	bGearOutMode                 :BOOL;
    fMasterSyncPosition           :LREAL;  
    fSlaveSyncPosition              :LREAL;  

	bReady                            :BOOL;  
    bStartSync		 	               :BOOL;	
	bInSync		 	                   :BOOL;	
    bBusy                               :BOOL;	
	bError				               :BOOL;		

END_STRUCT
END_TYPE

// ---- DUTs/06_Interface/FB_Interface/ST_RecY.TcDUT
TYPE ST_RecY : //
STRUCT
	bEnable		                        :BOOL;	
 
	bReady                            :BOOL;  
	bRecOK	 	                   :BOOL;	
	bError				               :BOOL;			
END_STRUCT
END_TYPE

// ---- DUTs/06_Interface/FB_Interface/ST_TenBuffer.TcDUT
TYPE ST_TenBuffer :  //张力FB 接口信号
STRUCT
   	bExecute			                        :BOOL;	
  

	bError                                       :BOOL;

	bReady                                      :BOOL;
	bStartSync		                             :BOOL;
	bInSync		                                 :BOOL;//同步状态

END_STRUCT
END_TYPE

// ---- DUTs/06_Interface/FB_Interface/ST_Tension_1.TcDUT
TYPE ST_Tension_1 :  //张力FB 接口信号
STRUCT
	fWindDiameter           :REAL;//放卷实时直径
    fDanserDegree           :REAL;//摆杆实时位置
   
   	bTenExecute		        :BOOL;	//张力使能
	bStudyExecute           :BOOL;  //摆杆学习开始     
   	fStudyDiameter          :REAL;  //摆杆学习时放卷直径
	
	bReady                    :BOOL;  //张力功能准备好
	bTensionOK		       :BOOL;	//张力使能OK

	bError			           :BOOL;	//张力出错
                         
END_STRUCT
END_TYPE

// ---- DUTs/06_Interface/Method/ST_Method.TcDUT
TYPE ST_Method :  //    方法
STRUCT

             AllTempTurnON                            :ST_MethodOut;//温控开
             AllTempTurnOFF                           :ST_MethodOut;//温控关
          
             AllRectLock                                  :ST_MethodOut;//纠偏外部锁定
             AllRectAuto                                  :ST_MethodOut;//纠偏自动
             AllRectManual                              :ST_MethodOut;//纠偏手动
             AllRectCenter                               :ST_MethodOut;//j纠偏居中

            // AllTen                                          :ST_MethodOut;
          

             AllGear                                        :ST_MethodOut;
             AllHome                                      :ST_MethodOut;


           // P1Ten                                             :ST_MethodOut;
           // P2Ten                                             :ST_MethodOut;
            //P3Ten                                             :ST_MethodOut;

            P1Pole                                            :ST_MethodOut;   
            P2Pole                                            :ST_MethodOut;   
            P3Pole                                            :ST_MethodOut;   
            P1GM                                             :ST_MethodOut;    
            P2GM                                             :ST_MethodOut;   


            P1CamIn                                        :ST_MethodOut;
            P2CamIn_U                                     :ST_MethodOut;
            P2CamIn_D                                     :ST_MethodOut;
            P3CamIn_U                                     :ST_MethodOut;
            P3CamIn_D                                     :ST_MethodOut;


          P4ShortTestHome                              :ST_MethodOut;  //短路测试
          P4StackHome                                    :ST_MethodOut; //叠片台
          P4CutSyncHome                                 :ST_MethodOut ;  //裁切同步
          P4NGHome                                       :ST_MethodOut ;  //NG料盒



END_STRUCT
END_TYPE

// ---- DUTs/06_Interface/Method/ST_MethodOut.TcDUT
TYPE ST_MethodOut :  //    方法
STRUCT
             Execute            :BOOL;  
             Done1               :BOOL;  
             Done2               :BOOL;  
             Error               :BOOL;

END_STRUCT
END_TYPE

// ---- DUTs/07_Name/ST_MotorName.TcDUT
TYPE ST_MotorName ://毛刷马达名称
STRUCT
	DDR_Dust:INT;//主驱辊除尘毛刷
	CuterBeltDust:INT;//裁切输送皮带除尘
	NGReverseBeltDust	:INT;//踢废倒装皮带除尘
	DedustBeltDust	:INT;//极片上表面除尘皮带除尘
	DedustReverseBeltDust	:INT;//极片下表面除尘倒装皮带除尘

   PoleBrushDust_U        :INT;     //极片上表面毛刷除尘**)
   PoleBrushDust_D        :INT;     //极片下表面毛刷除尘**)
   FeduanbeltDust1		  :INT;  //分段皮带1毛刷
   FeduanbeltDust2		  :INT;  //分段皮带2毛刷
   FeduanbeltDust3		  :INT;  //分段皮带3毛刷
   
END_STRUCT
END_TYPE

// ---- DUTs/07_Name/ST_NGMark.TcDUT
TYPE ST_NGMark :   //模切段NG标志位
STRUCT
	NGMark:ARRAY[1..30]	OF	BOOL	;	//[1]极片长度不良计数标志位,[2]极片宽度不良计数标志位,[3]R角不良计数标志位,[4]极耳不良计数标志位,[5]CIL宽不良计数标志位,[6]极片角度、边缘角度不良计数标志位,[7]尺寸其他不良,[8]接带不良计数标志位,[9]极片破损不良计数标志位,[10]划痕不良计数标志位,[11]亮斑不良计数标志位,[12]黑点不良计数标志位,[13]脏污不良计数标志位,[14]脱碳不良计数标志位,


	//NGMark[1]	:	BOOL	;	//	极片长度不良计数标志位
	//NGMark[2]	:	BOOL	;	//	极片宽度不良计数标志位
	//NGMark[3]	:	BOOL	;	//	R角不良计数标志位
	//NGMark[4]	:	BOOL	;	//	极耳不良计数标志位
	//NGMark[5]	:	BOOL	;	//	CIL宽不良计数标志位
	//NGMark[6]	:	BOOL	;	//	极片角度、边缘角度不良计数标志位
	//NGMark[7]	:	BOOL	;	//	尺寸其他不良
	//NGMark[8]	:	BOOL	;	//	接带不良计数标志位
	//NGMark[9]	:	BOOL	;	//	极片破损不良计数标志位
	//NGMark[10]	:	BOOL	;	//	划痕不良计数标志位
	//NGMark[11]	:	BOOL	;	//	亮斑不良计数标志位
	//NGMark[12]	:	BOOL	;	//	黑点不良计数标志位
	//NGMark[13]	:	BOOL	;	//	脏污不良计数标志位
	//NGMark[14]	:	BOOL	;	//	脱碳不良计数标志位




END_STRUCT
END_TYPE

// ---- DUTs/07_Name/ST_TableNo.TcDUT
TYPE ST_TableNo ://    凸轮表号
STRUCT
         Cuter	:UINT ;(*裁切切刀凸轮编号*)
		 CuterStop	:UINT ;(*裁切切刀停止凸轮编号*)
		 Mould	:UINT;(*模具切刀凸轮编号*)
		 MouldStop	:UINT;(*模具切刀停止凸轮编号*)
         Dirver	:UINT;(*主驱动凸轮编号*)
		 VirDirver:UINT;(*虚驱动凸轮编号*)
         VirBelt	:UINT;(*虚拟皮带凸轮编号*)
         NgPush	:UINT;(*NG踢料凸轮编号*)
		 NgPushStop	:UINT;(*NG踢料停止凸轮编号*)
         BufferLine	:UINT;(*极片缓存凸轮编号*)
		 CCDPress:UINT;(*CCD压片凸轮编号*)
		 BufferLine_1	:UINT;(*极片缓存凸轮编号*)
END_STRUCT
END_TYPE

// ---- DUTs/07_Name/ST_CylinderName.TcDUT
TYPE ST_CylinderName :   //气缸名称
STRUCT
Inflation_L	:INT;(*左放卷气胀轴气缸*)	
Inflation_R	:INT;(*右放卷气胀轴气缸*)	
BoardPressL	:INT;(*左接带压板气缸*)	
BoardPressR	:INT;(*右接带压板气缸*)	
DriverPressAux	:INT;(*辅助驱动压辊气缸*)	
CoderRollPress	:INT;(*编码器辊压辊气缸*)	
DriverPressDDR	:INT;(*主驱动压辊气缸*)	
NGRevBeltUpDown	:INT;(*踢废倒装皮带升降气缸*)	
NGRevBeltTension	:INT;(*踢废倒装皮带张紧气缸*)	
PoleBrushDustPush_U	:INT;(*极片上表面毛刷除尘升降缸*)	
PoleWindDustPush_U	:INT;(*极片上表面风刀除尘升降缸*)	
PoleBrushDustPush_D	:INT;(*极片下表面毛刷除尘升降缸*)	
PoleWindDustPush_D	:INT;(*极片下表面风刀除尘升降缸*)	
DustRevBeltUpDown	:INT;(*极片下表面除尘倒装皮带升降气缸*)	
NGBoxLock1	:INT;(*NG料盒归正气缸1*)	
NGBoxLock2	:INT;(*NG料盒归正气缸2*)	
WasteBoxPush	:INT;(*连续废料收集箱推料气缸*)	
END_STRUCT
END_TYPE

// ---- DUTs/07_Name/ST_VirAxisName.TcDUT
TYPE ST_VirAxisName :   //正极虚轴名称
STRUCT
 VirMain:INT;//模切虚拟主轴
 VirDriver:INT;//模切虚拟驱动辊
 VirBelt:INT;//模切虚拟皮带轴
  
END_STRUCT
END_TYPE

// ---- DUTs/06_Interface/FB_Interface/ST_Tension.TcDUT
TYPE ST_Tension :  //张力FB 接口信号
STRUCT
	fWindDiameter           :REAL;//放卷实时直径
    fDanserDegree           :REAL;//摆杆实时位置
   
   	bTenExecute		        :BOOL;	//张力使能
	bStudyExecute           :BOOL;  //摆杆学习开始     
   	fStudyDiameter          :REAL;  //摆杆学习时放卷直径
	
	bReady                    :BOOL;  //张力功能准备好
	bTensionOK		       :BOOL;	//张力使能OK

	bError			           :BOOL;	//张力出错
                         
END_STRUCT
END_TYPE

// ---- DUTs/09_保持型汇总/LocalProduction.TcDUT
TYPE  LocalProduction :
STRUCT
	OutFlag1:BOOL;(*产量计数标志1*)
	OutFlag2:BOOL;(*产量计数标志2*)
	NGFlag:ARRAY[1..50] OF BOOL;(*NG1计数标志*)

	RunFlag:BOOL;(*运行标志*)
	WaitFlag:BOOL;(*待料标志*)
	AlarmFlag:BOOL;(*故障标志*)
	DelDataAMBtn:BOOL;(*白班数据清除按钮*)
	DelDataPMBtn:BOOL;(*夜班数据清除按钮*)
	NowOutTotal:REAL;(*当前班次加工总数*)
	NowRate:REAL;(*当前班次良率*)
	HMI_NGClearAMBtn:ARRAY[1..50] OF BOOL;//白班NG类型计数清零
	HMI_NGClearPMBtn:ARRAY[1..50] OF BOOL;//夜班NG类型计数清零
	
//产能清零
	HMI_DelDataAMBtn			:BOOL;//白班产能清零
	HMI_DelDataPMBtn			:BOOL;//夜班产能清零
(*产能统计*)
	HMI_TodayTotal				:REAL;(*当天24H生产总数*)
	HMI_TodayOK					:REAL; (*当天24H生产OK总数*)
	HMI_TodayNG 				:REAL; (*当天24H生产NG总数*)
	
	HMI_HistoryTotal			:ARRAY[1..7 ] 	OF REAL ;(*历史每天24H生产总数ARRAY[1..7 ]*)
	HMI_HistoryOK				:ARRAY[1..7 ] 	OF REAL ;(*历史每天24H生产OK总数ARRAY[1..7 ]*)
	HMI_HistoryNG 				:ARRAY[1..7 ] 	OF REAL ; (*历史每天24H生产NG总数ARRAY[1..7 ]*)
	DayCountTotal				:REAL;(*白班产量合计*)
	NightCountTotal				:REAL;(*夜班产量合计*)
	SaveNowDay					:INT;
	SaveNowMonth				:INT;
	nDayRunTimeCnt				:ARRAY[8..19 ] 	OF UDINT;		(*白班运行时间统计*)
	nDayAlarmTimeCnt			:ARRAY[8..19 ] 	OF UDINT;		(*白班报警时间统计*)
	nDayWaitTimeCnt				:ARRAY[8..19 ] 	OF UDINT;		(*白班待料时间统计*)
	nNightRunTimeCnt			:ARRAY[0..23 ] OF UDINT;		(*夜班运行时间统计*)
	nNightAlarmTimeCnt			:ARRAY[0..23 ] OF UDINT;		(*夜班报警时间统计*)
	nNightWaitTimeCnt			:ARRAY[0..23 ] OF UDINT;		(*夜班待料时间统计*)
	HourTimeDayCount			:ARRAY[8..19 ] 	OF REAL;		(*白班每小时产量*)
	HourTimeNightCount			:ARRAY[0..23] 	OF REAL;		(*夜班每小时产量*)
	NgPerHourDayCount			:ARRAY[1..50 ] 	OF REAL;		(*白班1-30种类的不良分类*)
	NgPerHourNightCount			:ARRAY[1..50 ] 	OF REAL;		(*夜班1-30种类的不良分类*)
	HMI_TotalCount				:REAL;(*总产量*)
	HMI_OkCount					:REAL;(*OK产量*)
	HMI_NgCount					:REAL;(*Ng产量*)
	HMI_Qualified 				:REAL;(*良率*)
	HMI_NG_Qualified 			:REAL;(*不良率*)
	HMI_OEE							:REAL;//设备稼动率
	HMI_DayOkCount				:REAL;(*白班OK产量*)
	HMI_DayNgCount				:REAL;(*白班Ng产量*)
	HMI_DayQualified 			:REAL;(*白班良率*)
	HMI_DayNG_Qualified 		:REAL;(*白班不良率*)
	HMI_NightOkCount			:REAL;(*夜班OK产量*)
	HMI_NightNgCount			:REAL;(*夜班Ng产量*)
	HMI_NightQualified 			:REAL;(*夜班良率*)
	HMI_NightNG_Qualified 		:REAL;(*夜班不良率*)
	DayRunTimeTotal				:REAL;(*白班总运行时间合计*)
	NightRunTimeTotal			:REAL;(*夜班总运行时间合计*)
	DayAlarmTimeTotal			:REAL;(*白班总报警时间合计*)
	NightAlarmTimeTotal			:REAL;(*夜班总报警时间合计*)
	DayWaitTimeTotal			:REAL;(*白班总待料时间合计*)
	NightWaitTimeTotal			:REAL;(*夜班总待料时间合计*)
	RunTimeTotal				:REAL;(*总运行时间合计*)
	WaitTimeTotal				:REAL;(*总待料时间合计*)
	AlarmTimeTotal				:REAL;(*总报警时间合计*)
	(*历史数据变量汇总1-7天*)
	(*白班*)
	DayReadDayHistory			:ARRAY[1..7 ] 	OF INT;(*历史日*)
	DayReadMonthHistory			:ARRAY[1..7 ] 	OF INT;(*历史月*)
	DayCountTotalHistory		:ARRAY[1..7 ] 	OF REAL ;(*历史白班每天生产总数*)
	HMI_DayOkCountHistory		:ARRAY[1..7 ] 	OF REAL ;(*历史白班每天生产OK总数*)
	HMI_DayNgCountHistory		:ARRAY[1..7 ] 	OF REAL ;(*历史白班每天生产NG总数*)
	HMI_DayQualifiedHistory		:ARRAY[1..7 ] 	OF REAL ;  (*历史白班每天良率*)
	DayRunTimeTotalHistory		:ARRAY[1..7 ] 	OF REAL ;(*历史每天白板总运行时间合计*)
	DayWaitTimeTotalHistory		:ARRAY[1..7 ] 	OF REAL ;(*历史每天白板总待料时间合计*)
	DayAlarmTimeTotalHistory	:ARRAY[1..7 ] 	OF REAL ;(*历史每天白板总报警时间合计*)
	NgPerHourDayCountHistory	:ARRAY[1..7,1..50 ] 	OF REAL ;(*历史每天白班各类NG数量*)
	HourTimeDayCountHistory		:ARRAY[1..7,8..19 ] 	OF REAL ;(*历史每天白班每小时产量*)
	(*夜班*)
	NightCountTotalHistory		:ARRAY[1..7 ] 	OF REAL ;
	HMI_NightOkCountHistory		:ARRAY[1..7 ] 	OF REAL ;
	HMI_NightNgCountHistory		:ARRAY[1..7 ] 	OF REAL ;
	HMI_NightQualifiedHistory	:ARRAY[1..7 ] 	OF REAL ;
	NightRunTimeTotalHistory	:ARRAY[1..7 ] 	OF REAL ;
	NightWaitTimeTotalHistory	:ARRAY[1..7 ] 	OF REAL ;
	NightAlarmTimeTotalHistory	:ARRAY[1..7 ] 	OF REAL ;
	NgPerHourNightCountHistory	:ARRAY[1..7,1..50 ] 	OF REAL ;
	HourTimeNightCountHistory	:ARRAY[1..7,0..23] 	OF REAL ;
	(*历史数据变量汇总1-7天*)


(**********************************生产统计数据********************************************)
	DayRunTime_min:ARRAY[8..19] 	OF REAL;	(*白班每小时运行时间*)
	NightRunTime_min:ARRAY[0..23] 	OF REAL;	(*夜班每小时运行时间*)
	AllDayRunTime_min: REAL;	(*白班总运行时间*)
	AllNightRunTime_min: REAL;	(*夜班总运行时间*)

	DayWaitTime_min:ARRAY[8..19] 	OF REAL;	(*白班待料每小时时间*)
	NightWaitTime_min:ARRAY[0..23] 	OF REAL;	(*夜班待料每小时时间*)
	AllDayWaitTime_min: REAL;(*白班总待料时间*)
	AllNightWaitTime_min: REAL;(*夜班总待料时间*)

	DayAlmTime_min:ARRAY[8..19] 	OF REAL;	(*白班每小时报警时间*)
	NightAlmTime_min:ARRAY[0..23] OF REAL;	(*夜班每小时报警时间*)
	AllDayAlmTime_min: REAL;	(*白班总报警时间*)
	AllNightAlmTime_min: REAL;	(*夜班总报警时间*)

	DayBlockTime_min:ARRAY[0..23] 	OF REAL;(*白班每小时堵料时间*)
	NightBlockTime_min:ARRAY[0..23] 	OF REAL;(*夜班每小时堵料时间*)
	AllDayBlockTime_min: REAL;(*白班总堵料时间*)
	AllNightBlockTime_min: REAL;(*夜班总堵料时间*)
	
	HMINgClassCount_Day:ARRAY[1..50,0..23] 	OF REAL;(*白班每种NG类型每小时统计 ,,,NG类型，小时*)
	HMINgClassCount_Night:ARRAY[1..50,0..23] 	OF REAL;(*夜班每种NG类型每小时统计 ,,,NG类型，小时*)
	
	
	

	HisDayRunTime_min	:ARRAY[1..7,8..19 ] OF REAL ; (*历史白班每小时运行时间*)
	HisNightRunTime_min	:ARRAY[1..7,0..23 ] OF REAL ; (*历史夜班每小时运行时间*)
	HisAllDayRunTime_min:ARRAY[1..7] OF REAL ;	(*历史白班总运行时间*)
	HisAllNightRunTime_min:ARRAY[1..7 ] OF REAL ;	(*历史夜班总运行时间*)

	HisDayWaitTime_min	:ARRAY[1..7,8..19 ] OF REAL ; (*历史白班每小时待料时间*)
	HisNightWaitTime_min:ARRAY[1..7,0..23 ] OF REAL ; (*历史夜班每小时待料时间*)
	HisAllDayWaitTime_min:ARRAY[1..7] OF REAL ;	(*历史白班总待料时间*)
	HisAllNightWaitTime_min:ARRAY[1..7 ] OF REAL ;	(*历史夜班总待料时间*)

	HisDayAlmTime_min	:ARRAY[1..7,8..19 ] OF REAL ; (*历史白班每小时报警时间*)
	HisNightAlmTime_min	:ARRAY[1..7,0..23 ] OF REAL ; (*历史夜班每小时报警时间*)
	HisAllDayAlmTime_min:ARRAY[1..7] OF REAL ;	(*历史白班总报警时间*)
	HisAllNightAlmTime_min:ARRAY[1..7 ] OF REAL ;(*历史夜班总报警时间*)

	HisHMINgClassCount_Day:ARRAY[1..50,0..23,1..7] 	OF REAL;(*历史白班每种NG类型每小时统计,,,NG类型，小时，天*)
	HisHMINgClassCount_Night:ARRAY[1..50,0..23,1..7] 	OF REAL;(*历史夜班每种NG类型每小时统计,,,NG类型，小时，天*)

	
	HMI_TodayNGQualified:ARRAY[1..50] OF REAL;//当天白班各种NG类型NG率
	HMI_NightNGQualified:ARRAY[1..50] OF REAL;//当天夜班各种NG类型NG率	
	
	HMI_HisTodayNGQualified:ARRAY[1..50,1..7] OF REAL;//历史白班各种NG类型NG率
	HMI_HisNightNGQualified:ARRAY[1..50,1..7] OF REAL;//历史夜班各种NG类型NG率
	
END_STRUCT
END_TYPE

// ---- DUTs/09_保持型汇总/ST_Data.TcDUT
TYPE ST_Data :
STRUCT
	 AnBeltData:ARRAY[1..40]   OF  ST_BeltData;//正极皮带数据
	 CaBeltData:ARRAY[1..40]   OF  ST_BeltData;//负极皮带数据
	AnTabData:ARRAY[1..20]   OF  ST_TabData;//正极极耳数据
	CaTabData:ARRAY[1..20]   OF  ST_TabData;//负极极耳数据
	AnIntervalData:ARRAY[1..20]   OF  ST_IntervalData;//正极极耳间距数据
	CaIntervalData:ARRAY[1..20]   OF  ST_IntervalData;//负极极耳间距数据
	AnOffsetData:ARRAY[1..50]   OF  REAL;//正极主驱补偿数据
	CaOffsetData:ARRAY[1..50]   OF  REAL;//负极主驱补偿数据
	
	AnYellowPos:ARRAY [1..100] OF REAL;//正极黄标位置
	CaYellowPos:ARRAY [1..100] OF REAL;//负极黄标位置
	AnYellowMark:ARRAY [1..100] OF BOOL;//正极黄标标志--给到极片
	CaYellowMark:ARRAY [1..100] OF BOOL;//负极黄标标志--给到极片
	
	AnTapePos:ARRAY [1..100] OF REAL;//正极接带位置
	CaTapePos:ARRAY [1..100] OF REAL;//负极接带位置
	AnTapeMark:ARRAY [1..100] OF BOOL;//正极接带标志--给到极片
	CaTapeMark:ARRAY [1..100] OF BOOL;//负极接带标志--给到极片
	
	
	AnYellowJump_R:ARRAY [1..100] OF BOOL;//极片黄标R角跳切标志
	AnYellowJump_C:ARRAY [1..100] OF BOOL;//极片黄标裁切跳切标志
	AnTapeJump_R:ARRAY [1..100] OF BOOL;//极片接带R角跳切标志
	AnTapeJump_C:ARRAY [1..100] OF BOOL;//极片接带裁切跳切标志
	
	CaYellowJump_R:ARRAY [1..100] OF BOOL;//极片黄标R角跳切标志
	CaYellowJump_C:ARRAY [1..100] OF BOOL;//极片黄标裁切跳切标志
	CaTapeJump_R:ARRAY [1..100] OF BOOL;//极片接带R角跳切标志
	CaTapeJump_C:ARRAY [1..100] OF BOOL;//极片接带裁切跳切标志
			
END_STRUCT
END_TYPE

// ---- DUTs/09_保持型汇总/ST_Name.TcDUT
TYPE ST_Name :
STRUCT
(**轴**)
	AnAxisNo:      ST_AxisName;  //正极
	CaAxisNo:      ST_AxisName;//负极
	
    AnVirAxisNo:      ST_VirAxisName;//正极
	CaVirAxisNo:      ST_VirAxisName;//负极
	VirTimeWind:INT;//模切虚拟摆杆放卷轴 
(**气缸**)
	AnCYNo:        ST_CylinderName;//正极
	CaCYNo:        ST_CylinderName;//负极

(**电磁阀**)
	AnEVNo:        ST_ElectValveName;//正极
	CaEVNo:        ST_ElectValveName;//负极

(***纠偏**)
    AnRecNo:         ST_RecName;//正极
	CaRecNo:         ST_RecName;//负极

(***凸轮表号**)
	 AnTableNo:  ST_TableNo;// 正极
	 CaTableNo:  ST_TableNo;// 负极
	 
(***除尘电机号**)
	 AnMotorNo:  ST_MotorName;// 正极
	 CaMotorNo:  ST_MotorName;// 负极

(***数据工位号**)	 
	 AnBeltNo:ST_BeltNo;//正极
	 CaBeltNo:ST_BeltNo;//负极
	 AnTabNo:ST_TabNo;//正极
	 CaTabNo:ST_TabNo;//负极
	 AnIntervalNo:ST_IntervalNo;//正极
	 CaIntervalNo:ST_IntervalNo;//负极
END_STRUCT
END_TYPE

// ---- DUTs/09_保持型汇总/ST_Parameter.TcDUT
TYPE ST_Parameter :
STRUCT
	FanEn:BOOL;//风速仪屏蔽
	MaFanEn:BOOL;//风机平板
	AnPar: ST_ParProduct;   //正极工艺参数
	CaPar: ST_ParProduct;   //负极工艺参数
	parPublic:ST_PARpublic;//公共工艺参数
	
	parFilterAD            :ARRAY[1..MaxAINo] OF ST_ParFilterAD;
	parFilterDA            :ARRAY[1..2] OF ST_ParFilterDA;
	
	parDA                   :ARRAY[1..8] OF INT;   //模拟量输出
	iModeEN :                     IModeEN;//功能屏蔽

	  ////////////////////////////////////////////////////////////////////////////////////////////////////////////////断电保持中转变量////////////////////////////////////////////////////////////////////// 
	   	   
	 PoleData:ST_Data;	   
	   
	aAnDay_date: Day_date; //正极产能；
	aCaDay_date: Day_date; //负极产能；
	cCn_An:REAL;
	cCn_Ca:REAL;
		 
 	 YL_GVL2: ARRAY [1..60] OF DINT ;//内部预留；//  1、正极R角已经切的次数;  2、正极R角设置清废报警次数；3、负极R角已经切的次数;  4、负极R角设置清废报警次数；
	
(*产能统计*)	
	HMI_AnTodayNGClass_AM		:ARRAY[1..30 ] 	OF REAL;(*当天白班各类NG数量ARRAY[1..30 ]-----正极*)
	HMI_AnTodayNGClass_PM		:ARRAY[1..30 ] 	OF REAL;(*当天夜班各类NG数量ARRAY[1..30 ]-----正极*)
	HMI_AnTodayNG_AM:REAL;(*当天白班生产NG总数-----正极*)
	HMI_AnTodayNG_PM:REAL;(*当天夜班生产NG总数-----正极*)
	
	HMI_CaTodayNGClass_AM		:ARRAY[1..30 ] 	OF REAL;(*当天白班各类NG数量ARRAY[1..30 ]-----负极*)
	HMI_CaTodayNGClass_PM		:ARRAY[1..30 ] 	OF REAL;(*当天夜班各类NG数量ARRAY[1..30 ]-----负极*)
	HMI_CaTodayNG_AM:REAL;(*当天白班生产NG总数-----负极*)
	HMI_CaTodayNG_PM:REAL;(*当天夜班生产NG总数-----负极*)
	
	  iTargetTorque	                    	:ARRAY[1..2]OF INT;			                     (*单位为0.1%*) //最大为100

	CleanTimeHMIHour1:INT;//白班第一次清洁时间Hour\
	CleanTimeHMIMin1:INT;//白班第一次清洁时间Min
	CleanTimeHMIHour2:INT;//白班第二次清洁时间Hour
	CleanTimeHMIMin2:INT;//白班第二次清洁时间Min
	CleanTimeHMIHour3:INT;//夜班第一次清洁时间Hour
	CleanTimeHMIMin3:INT;//夜班第一次清洁时间Min
	CleanTimeHMIHour4:INT;//夜班第二次清洁时间Hour
	CleanTimeHMIMin4:INT;//夜班第二次清洁时间Ming
	CibangTimeHMIHour1:INT;//正极磁棒校验到期时间Hour
	CibangTimeHMIDay1:INT;//正极磁棒校验到期时间日
	CibangTimeHMIHour2:INT;//负极磁棒校验到期时间Hour
	CibangTimeHMIDay2:INT;//负极磁棒校验到期时间日	
	BrushTimeHMIHour1:INT;//正极毛刷清洁时间Hour
	BrushTimeHMIDay1:INT;//正极毛刷清洁时间Day
	BrushTimeHMIHour2:INT;//负极毛刷清洁时间Hour
	BrushTimeHMIDay2:INT;//负极毛刷清洁时间Day

(*****************************************************极耳基准20240101SJ*********************************************************************)	  

	bCompSel:BOOL;//补偿方案选择		
	
(***************************************************线扫20240219***********************************************************************)
	iLineScanSel:BOOL;//线扫结果控制模式
	
	  
(***************************************************4l连续黄标尾料检测***********************************************************************)
	fYellowMackLength1           :REAL;// 相邻黄标后边距离	
	  
END_STRUCT
END_TYPE

// ---- DUTs/30_Parameter/ST_DT_To_MQ_MES.TcDUT
TYPE ST_DT_To_MQ_MES  :
STRUCT
//PC写给PLC的-----先下发给叠台，叠台再和模切做通讯-------需要上料时PLC往该地址写入Error
PostiveCode1				:STRING(49);//正极左1条码		1
PostiveCode2				:STRING(49);//正极右2条码		2
NegativeCode1				:STRING(49);//负极左1条码		3
NegativeCode2				:STRING(49);//负极右2条码		4
Station1_Code				:STRING(49);//叠台1隔膜条码		5
Station2_Code				:STRING(49);//叠台2隔膜条码		6
Station3_Code				:STRING(49);//叠台3隔膜条码		7
Station1_BlueCode			:STRING(49);//叠台1l蓝胶条码		8
Station2_BlueCode			:STRING(49);//叠台2蓝胶条码		9
Station3_BlueCode			:STRING(49);//叠台3蓝胶条码		10
CellCode					:STRING(49);//后段二维码胶条码	11
BlueCode					:STRING(49);//后段蓝胶条码		12

//MES条码校验信号交互----PC_To_PLC
Mes_PcToPlc1:        BOOL;   //正极左1条码条码校验完成信号
Mes_PcToPlc2:        BOOL;   //正极右2条码校验完成信号
Mes_PcToPlc3:        BOOL;   //负极左1条码	校验完成信号
Mes_PcToPlc4:        BOOL;   //负极右2条码校验完成信号
Mes_PcToPlc5:        BOOL;   //叠台1隔膜条码校验完成信号
Mes_PcToPlc6:        BOOL;   //叠台2隔膜条码校验完成信号
Mes_PcToPlc7:        BOOL;   //叠台3隔膜条码校验完成信号
Mes_PcToPlc8:        BOOL;   //叠台1l蓝胶条码校验完成信号
Mes_PcToPlc9:        BOOL;   //叠台2蓝胶条码校验完成信号
Mes_PcToPlc10:        BOOL;  //叠台3蓝胶条码校验完成信号
Mes_PcToPlc11:        BOOL;   //后段二维码胶条码校验完成信号
Mes_PcToPlc12:        BOOL;   //后段蓝胶条码校验完成信号	

//MES条码校验信号交互----PLC_To_PC
MesClear_Pc1:        BOOL;   //正极左1换料信号清理
MesClear_Pc2:        BOOL;   //正极右2换料信号清理
MesClear_Pc3:        BOOL;   //负极左1换料信号清理
MesClear_Pc4:        BOOL;   //负极右2换料信号清理

END_STRUCT
END_TYPE

// ---- DUTs/30_Parameter/ST_MouldRecY.TcDUT
TYPE ST_MouldRecY :
STRUCT
		fRecBaseValue1                         :REAL:=5;//模具Y纠偏传感器基准值1(靠近大板)
		fRecBaseValue2							:REAL:=5;//模具Y纠偏传感器基准值2(远离大板)	
		fRectifyCoe                                 :REAL:=1;//纠偏系数	
		bRectifyDir                                 :BOOL;//纠偏方向
		fRecBaseRange                           :REAL:=0.2;//纠偏无效范围     注：纠偏量超出此值，才会进行动作。
		iMode                                        :INT:=1;//纠偏模式   1=单边纠偏；2=双边纠偏
		fRecAxisPos_H                             :REAL:=4;//纠偏电机上限
		fRecAxisPos_L                             :REAL:=4;//纠偏电机下限
END_STRUCT
END_TYPE

// ---- DUTs/30_Parameter/ST_MQ_To_DT_MES.TcDUT
TYPE ST_MQ_To_DT_MES  :
STRUCT
//PC写给PLC的-----先下发给叠台，叠台再和模切做通讯-------需要上料时PLC往该地址写入Error
PostiveCode1				:STRING(49);//正极左1条码		1
PostiveCode2				:STRING(49);//正极右2条码		2
NegativeCode1				:STRING(49);//负极左1条码		3
NegativeCode2				:STRING(49);//负极右2条码		4
Station1_Code				:STRING(49);//叠台1隔膜条码		5
Station2_Code				:STRING(49);//叠台2隔膜条码		6
Station3_Code				:STRING(49);//叠台3隔膜条码		7
Station1_BlueCode			:STRING(49);//叠台1l蓝胶条码		8
Station2_BlueCode			:STRING(49);//叠台2蓝胶条码		9
Station3_BlueCode			:STRING(49);//叠台3蓝胶条码		10
CellCode					:STRING(49);//后段二维码胶条码	11
BlueCode					:STRING(49);//后段蓝胶条码		12

//MES条码校验信号交互----PC_To_PLC
Mes_PcToPlc1:        BOOL;   //正极左1条码条码校验完成信号
Mes_PcToPlc2:        BOOL;   //正极右2条码校验完成信号
Mes_PcToPlc3:        BOOL;   //负极左1条码	校验完成信号
Mes_PcToPlc4:        BOOL;   //负极右2条码校验完成信号
Mes_PcToPlc5:        BOOL;   //叠台1隔膜条码校验完成信号
Mes_PcToPlc6:        BOOL;   //叠台2隔膜条码校验完成信号
Mes_PcToPlc7:        BOOL;   //叠台3隔膜条码校验完成信号
Mes_PcToPlc8:        BOOL;   //叠台1l蓝胶条码校验完成信号
Mes_PcToPlc9:        BOOL;   //叠台2蓝胶条码校验完成信号
Mes_PcToPlc10:        BOOL;  //叠台3蓝胶条码校验完成信号
Mes_PcToPlc11:        BOOL;   //后段二维码胶条码校验完成信号
Mes_PcToPlc12:        BOOL;   //后段蓝胶条码校验完成信号	

//MES条码校验信号交互----PLC_To_PC
Mes_PlcToPc1:        BOOL;   //正极左1换料信号
Mes_PlcToPc2:        BOOL;   //正极右2换料信号
Mes_PlcToPc3:        BOOL;   //负极左1换料信号
Mes_PlcToPc4:        BOOL;   //负极右2换料信号

END_STRUCT
END_TYPE

// ---- DUTs/30_Parameter/ST_ParFilterAD.TcDUT
TYPE ST_ParFilterAD :  //P1部分参数
STRUCT
	iLimitH             :REAL;//转换前高限值
	iLimitL             :REAL;//转换前低限值
	fRangeH         :REAL;//量程高限
	fRangeL          :REAL;//量程低限
	Out_Value        :REAL;//转换后

END_STRUCT
END_TYPE

// ---- DUTs/30_Parameter/ST_ParFilterDA.TcDUT
TYPE ST_ParFilterDA :  //P1部分参数
STRUCT
	X0:REAL;  //料带张力低限值g
	Y0:REAL;  //低限对应DA输出值
	X1:REAL; //料带张力高限值g
	Y1:REAL;//低限对应DA输出值
	bMode: BOOL;  //标定模式   TRUE为标定模式    
	iDAValue:REAL;//比例阀给定值     标定用
END_STRUCT
END_TYPE

// ---- DUTs/30_Parameter/ST_ParMachine.TcDUT
TYPE ST_ParMachine ://机械参数
STRUCT
       fMQDriverDiameter            :REAL:=71.62   ;//模切主驱辊直径
       fCuterDegDiameter				:REAL:=281.5   ;//裁切角度纠偏旋转半径
       fAuxDriverInDiameter         :REAL:=80   ;  //辅驱辊直径
	   fBelt1Scaling                      :REAL:=1   ;  //裁切皮带定长比例系数
	   fBelt2Scaling                      :REAL:=1   ;  //踢废倒装皮带定长比例系数
	   fBelt3Scaling                      :REAL:=1   ;  //上表面除尘皮带定长比例系数
	   fBelt4Scaling                      :REAL:=1   ;  //下表面除尘倒装皮带定长比例系数
	   fBelt5Scaling                      :REAL:=1   ;  //送料分段皮带1定长比例系数	   
	   fBelt6Scaling                      :REAL:=1   ;  //送料分段皮带2定长比例系数	   
	   fBelt7Scaling                      :REAL:=1   ;  //送料分段皮带3定长比例系数	  	   
//叠片主驱动  70
//叠片辅驱动  30
//NG皮带 46































END_STRUCT
END_TYPE

// ---- DUTs/30_Parameter/ST_MoQiePar.TcDUT
TYPE ST_MoQiePar :  //模切部分参数
STRUCT
(***张力参数*)
	TenCcw_WindL                            :BOOL;  //左放卷放卷方向
	TenCcw_WindR                            :BOOL;  //右放卷放卷方向
	bWindSelect								:BOOL;//放卷选择ON=使用左放卷
	WindPidSwitch                         :BOOL;  //放卷PID使能开关
	WindTenMinPos                      :REAL;//放卷摆杆最小角度
	WindTenMaxPos                     :REAL; //放卷摆杆最大角度
	WindTenBlancePos                  :REAL ;//放卷摆杆平衡角度
	WindTenTable                        :ARRAY[0..105,1..2]OF REAL;	//放卷摆杆采样数据
	
	TenCcw_AuxDriver                            :BOOL;  //辅驱放卷方向
	AuxDriverPidSwitch                         :BOOL;  //辅驱PID使能开关
	AuxDriverTenMinPos                      :REAL;//辅驱摆杆最小角度
	AuxDriverTenMaxPos                     :REAL; //辅驱摆杆最大角度
	AuxDriverTenBlancePos                  :REAL ;//辅驱摆杆平衡角度
	AuxDriverTenTable                        :ARRAY[0..105,1..2]OF REAL;	//辅驱摆杆采样数据		
	
	BufferPidSwitch                         :BOOL;  //缓存PID使能开关
	BufferMinPos                            :REAL;//缓存最小角度
	BufferMaxPos                           :REAL; //缓存最大角度
	BufferBlancePos                        :REAL ;//缓存平衡角度


   
END_STRUCT
END_TYPE

// ---- DUTs/30_Parameter/ST_ParProduct.TcDUT
TYPE ST_ParProduct ://工艺参数
STRUCT
(***HMI***)
	fYellowWidth :REAL:=25 ;    //黄标宽度
	fTapeWidth :REAL:=30 ;    //接带胶纸宽度
	fPoleWidth                          		  :REAL:=100 ;    //片宽
	fBeltSpacePos            :REAL:=280;//皮带运行定长
	
	//fCentreWidth_L								:REAL;//极耳中心_极片左侧宽度基准（程序内称左肩宽）
	//fCentreWidth_R								:REAL;//极耳中心_极片右侧宽度基准（程序内称右肩宽）
	fBlue_Mould                                :REAL;//蓝胶检测到模具倒角前的距离
	//iMould_Cuter                               :INT;//模具与裁切间的极耳个数
	fLineNG_Mould							   :REAL;//缺陷NG点到模具倒角前的距离
	bEarCheckMode                            :BOOL;   //极耳检测模式     FALSE:定长     TRUE：检测极耳
	fEarCheckLength                            :REAL;   //检测到极耳后走定长长度
	
	
	fFr_TenValuehmi									:REAL;//后摆杆张力比例阀大小HMI设置   单位%   范围：0-100
	fPressDDRhmi									:REAL;//主驱压辊比例阀大小HMI设置   单位%   范围：0-100
	
	iMouldCount1									:DINT;//前模具切刀计数
	iMouldCount2									:DINT;//后模具切刀计数
	iCuterCount									:DINT;//裁切切刀计数
	iMouldclear1                                 :BOOL;//前倒角模具切刀清零
	iMouldclear2                                 :BOOL;//后倒角模具切刀清零
	iCuterclear                                 :BOOL;//裁切切刀清零
	iMouldCountAlarm1						    :DINT;//前模具切刀计数报警
	iMouldCountAlarm2						    :DINT;//后模具切刀计数报警
	iCuterCountAlarm						     :DINT;//裁切切刀计数报警
	iCuterCountWarning							:DINT;//裁切切刀计数预警
	iCuterBarCode								:STRING(49);//切刀条码
	iReplaceCuterTime							:STRING(49);//换刀时间
	
	iMainVel                                  :UINT:=10;  //设置速度 PPM (最小值1,最大值200)          
	fMainHmiVel                                  :REAL;  //显示料带速度 M/min  
	fDiameterWarn_L:REAL;//左放卷卷径临界设置(警告)
	fDiameterWarn_R:REAL;//右放卷卷径临界设置(警告)
	fDiameterAlarm_L:REAL;//左放卷卷径临界设置(报警)
	fDiameterAlarm_R:REAL;//右放卷卷径临界设置(报警)
	
	MQ:ST_MoQiePar; (******放卷部分参数******)
	Rec:ST_MouldRecY;(******Y纠偏部分参数******)
	Machine: ST_ParMachine;   //机械参数常量   不允许外部改变
/////////////////////////////////////////////////////////////////////////////////////////////////CCD  R角闭环纠偏参数/////////////////////////////////////////////////////////////////////		
	Databace_R3:REAL;//CCD_R3 非极耳侧纵深基准正极5.6  负极2.6
	Databace_R4:REAL;//CCD_R4非极耳侧纵深基准正极5.6  负极2.6
	IntervalNum:UINT:=7; //片间距
	KI_Riao:REAL:=0.3;//比例系数		
	Limt_Max:REAL:=0.5; //最大补偿值
	Limt_Min:REAL:=-0.5;//最小补偿值
	TabSitebace:REAL;//基准肩宽
	TabWidthBace: REAL;//标准间距		
	AddAlarm:INT;
////////////////////////////////////////////////////////////////////////////////////////////////////////////////////////////////////////////////////////////////////////////////////////////////////		
(***内部使用**)
	fPoleWithOffset						:REAL; //主驱片宽补偿值（计算后）
	fMouldX_Offset						:REAL; //模具肩宽补偿值（计算后）
	fDegreeRectify						:REAL; //裁切角度纠偏值（计算后）
	fMouldY_Rectify						:REAL; //倒角深度纠偏值（计算后）
	
	
	fTension   							:REAL;//模切张力
	fSpeed								:REAL;//模切速度

//皮带齿轮比计算
	BeltDust1Great:REAL;//皮带1齿轮比计算系数
	BeltDust2Great:REAL;//皮带2齿轮比计算系数
	BeltDust3Great:REAL;//皮带3齿轮比计算系数

      

//新黄标、接带检测
	fLugBreadth:REAL:=59;//极耳宽度
	fCutBreadth:REAL:=22;//极耳边到切刀切点宽度---23.5+-1
	fYellowBreadth:REAL:=35;//黄标宽度
	fTapeBreadth:REAL:=35;//接带宽度
	
//初始卷径标定 ----demarcate
	rRoll_L:REAL:=1000;//缓存极片总长度(mm)
	rRollStartView:REAL;//放卷开始角度
        rRollFinishView:REAL;//放卷结束角度 
	rRollView :REAL;//放卷运动总角度  
	rRollDia:REAL;//初始卷径(计数输出)
	bDemarcateBtn:BOOL;//标定开始按钮

fTape_Mould                                :REAL;//接带检测到模具倒角前的距离	
fTape1_2                                :REAL;//前接带检到后接带检测的距离
(*****************************************************极耳基准20240101SJ*********************************************************************)	  

	fTabWidth: REAL;//极耳标准宽
	fDriverStanderBasePos: REAL;//极耳下降沿基准主驱凸轮位置
	fReadDriverPos3: REAL;//读取极耳下降沿主驱凸轮表位置
	bDriverStanderBasePosEN: BOOL;  //极耳大范围调整屏蔽	
	


END_STRUCT
END_TYPE

// ---- DUTs/30_Parameter/ST_ParPublic.TcDUT
TYPE ST_ParPublic :
STRUCT
		   fMainPos                   :REAL:=250;     //主轴关键点角度
		   //fBeltSpacePos            :REAL:=280;//皮带运行定长
END_STRUCT
END_TYPE

// ---- DUTs/30_Parameter/ST_ParTemperature.TcDUT
TYPE ST_ParTemperature ://   温控相关参数
STRUCT
   fTempSet                                   :REAL;// 设定温度温度(转换后)
   fTempOffset                               :REAL;// 设定温度温度(转换后);// 温度偏移

   fTempMax                                :REAL;     //温度高限设置

  fTempArea                               :REAL;     

END_STRUCT
END_TYPE

// ---- DUTs/31_其他辅助/ST_Timedata_2.TcDUT
TYPE ST_Timedata_2 :
STRUCT
	
	RunTime:ARRAY[0..25] OF UINT;//运行时间
    WaitTime:ARRAY[0..25] OF UINT;//待机时间
    AlmTime:ARRAY[0..25] OF UINT;//报警时间 	
    changeTime:ARRAY[0..25] OF UINT;//极片更换等待时间  	

	
END_STRUCT
END_TYPE

// ---- DUTs/32_系统/ST_SystemPart.TcDUT
TYPE ST_SystemPart ://系统功能块UDT
STRUCT
(***btn***)
	 btnStart                      :BOOL;  //面板启动
     btnStop                      :BOOL;  //面板停止
	 btnReset                     :BOOL;  //面板复位
     btnAuto                      :BOOL;//面板true=自动；false=手动
	 btnEstop                    :BOOL;//面板急停	 
	 
	 boStartLight                     :BOOL;           (***面板启动按钮灯***)
	 boResetLight                     :BOOL;           (***面板复位按钮灯***)
	 boStopLight                     :BOOL;           (***面板停止按钮灯***)
(***HMI*) 
	 hmiTenAll                    :BOOL;  //一键张力耦合
	 hmiDisTenAll                    :BOOL;  //一键张力解耦
	 hmiCamAll                    :BOOL;  //一键凸轮耦合
	 hmiDisCamAll                    :BOOL;  //一键凸轮解耦
	 hmiGoHome					:BOOL;//一键初始化(回原)
	 hmiClearBelt                 :BOOL;//一键清皮带(清除皮带上的料)
	 
	 hmiMQDriverOnce          :BOOL;  //模切驱动一片
	 hmiMQCutOnce             :BOOL;  //模切裁切一片 
	 
	 
(**Status**)
	 Homed						:BOOL;//初始化完成
	 Homeing					:BOOL;//初始化进行中
     Autoing                     :BOOL;   //自动运行中
	 Manuling                   :BOOL;  //手动运行中
	 Stoping                     :BOOL;   //停止中
	 Alarming                   :BOOL;   //报警中
	 bErrorStop                :BOOL;//报警停机

     bAutoCondition1         :BOOL;//自动准备好(初步)
	 bAutoCondition2         :BOOL;//自动准备好(张力凸轮OK)
     bStopFinished            :BOOL;
	 bAutoTen                  :BOOL;//自动允许气缸/张力/凸轮动作
	 bAutoMain                  :BOOL;//自动允许主轴动作
(***INIT***)
	hmiInit                        :BOOL;
    bInit                        :BOOL;
    bInitDone                :BOOL;
	bIniting                   :BOOL;
	
//条码校验OK	
	PolePieceNumberOK1   : BOOL;   //左料卷料号OK
	PolePieceNumberOK2   : BOOL;   //右料卷料号OK
END_STRUCT
END_TYPE

// ---- DUTs/33_M2/ST_BeltData.TcDUT
TYPE ST_BeltData ://皮带数据（裁断后）
STRUCT
	bHavePole   :BOOL;  //是否有极片
	iPanoramaNG:INT;//尺寸检测状态  1:OK  2:NG   3:无极片    0:无效
	iJumpCutNG:INT;//跳切连续NG  1:OK  2:NG  0:无效
	fPoleWidth:REAL;//片宽
	fPoleHeigh:REAL;//片高
	stPoleNo:STRING(256);//极片编号
 // fbST_CCDComSize:ST_CCDComSize;
	fTabWidth:REAL;  //尺寸检测CCD结果(极耳宽度)
	fTabHeigh:REAL;  //尺寸检测CCD结果(极耳高度)
	fTabSite   : REAL; // 极耳左，右边距(就是极耳位置，不分左右)
	//fOffsetDeg:REAL; //尺寸检测CCD结果(极片裁切面角度偏移)
	RoundedSize1                                :        REAL        ;//        圆角尺寸1 面积   叠片侧(正极)       负极相反
	RoundedSize2                                :        REAL        ;//         圆角尺寸2 面积    切刀侧(正极)        负极相反
	RoundedSize3                                :        REAL        ;//         圆角尺寸3纵深 叠片侧(正极)        负极相反
	RoundedSize4                                :        REAL        ;//        圆角尺寸4纵深 切刀侧(正极)     负极相反
	RoundedSize5                                :        REAL        ;//        圆角尺寸5 横深
	RoundedSize6                                :        REAL        ;//        圆角尺寸6横深
	RoundedSize7                                :        REAL        ;//      圆角尺寸7横深 叠片侧(正极)     负极相反
	RoundedSize8                               :        REAL        ;//        圆角尺寸8横深 切刀侧(正极)     负极相反
	PolePlateAngle1                                :        REAL        ;//        极片角度1  极片角度
	PolePlateAngle2                                :        REAL        ;//        极片角度2
	PolePlateAngle3                                :        REAL        ;//        极片角度3
	PolePlateAngle4                                :        REAL        ;//        极片角度4
	fPoleNGSizeNo:REAL;  //尺寸检测CCD结果(NG分类编号)
	iTabNGSizeNo:INT;  //尺寸检测CCD极耳抓边异常分类     1： OK  2: 极片抓边异常    3:极耳抓边异常     4：都抓边异常     5：极片或极耳角度异常    
	
	iPoleRAngleNG:INT;//尺寸检测CCD结果(R角NG)
	iFinish:INT;  //尺寸检测CCD结果指示(1=完成;2=NG;3=无片;0=无效)  SizeResults
	AppearanceResult:INT;// 极片外观判定结果   线扫NG、OK

	UnreelingTension                        :        REAL        ;//        放卷张力
	SlicingSpeed                                :        REAL        ;//        切片速度
	PolePlateLenth                                :        REAL        ;//        极片长度（走带方向）
	fPoleNGSacnNo:REAL;  //极片先扫NG编号(NG分类编号)
	
	bYellowMark:BOOL;//黄标标志--TRUE为黄标
	bBlueMark:BOOL;//接带标志--TRUE为接带
	Code				:STRING(49);//料卷条码
END_STRUCT
END_TYPE

// ---- DUTs/33_M2/ST_TabData.TcDUT
TYPE ST_TabData ://极耳数据（裁断前）
STRUCT
	fTab_OffsetM:					REAL;//倒角极片偏移量
	//fTabC_OffsetM:					REAL;//倒角前极耳中心偏移量
	//fTabR_OffsetM:					REAL;//倒角前极耳右侧偏移量
	fPhotoPosM:                 REAL;//倒角前拍照位置
	fTab_OffsetC:					REAL;//裁切前极片偏移量
	//fTabC_OffsetD:					REAL;//裁切前极耳中心偏移量
	//fTabR_OffsetD:					REAL;//裁切前极耳右侧偏移量
	fPhotoPosC:                 REAL;//裁切前拍照位置
	bCCDed_M:                  BOOL;//true:经过倒角CCD拍照标志
	bCCDed_C:                  BOOL;//true:经过裁切CCD拍照标志
	bTabOffsetNG_M:                  BOOL;//true:倒角CCD纠偏量超差标志
	bTabOffsetNG_C:                  BOOL;//true:裁切CCD纠偏量超差标志
	
	//bYellowMark:BOOL;//黄标标志--TRUE为黄标
	//bBlueMark:BOOL;//接带标志--TRUE为接带
	fTab_OffsetY   :REAL;//倒角极片偏移量Y  
	
	
END_STRUCT
END_TYPE

// ---- DUTs/33_M2/ST_AlarmWarn.TcDUT
TYPE ST_AlarmWarn :
STRUCT
	arrTenAlarm                                 :ARRAY[1..15]  OF BOOL;                  //张力报警
	arrCreatTableAlarm                         :ARRAY[1..30]  OF BOOL;             //创建凸轮报警
	arrCamInAlarm                               :ARRAY[1..30]  OF BOOL;             //凸轮耦合报警
	arrGearAlarm                                  :ARRAY[1..25]  OF BOOL;             //齿轮报警
	arrFlowAlarm                                  :ARRAY[1..50]  OF BOOL;             //流程报警
	arrLightWarn                                  :ARRAY[1..50]  OF BOOL;             //轻型警告(提示)
	arrRecAlarm                                 :ARRAY[1..15]  OF BOOL;                  //纠偏报警
END_STRUCT
END_TYPE

// ---- DUTs/33_M2/ST_BeltNo.TcDUT
TYPE ST_BeltNo ://皮带工位号（裁断后）
STRUCT
First	:INT:=1;		//	首片数据
OverHang	:INT:=2;		//	尺寸检测工位
NGBox1	:INT:=4;		//	踢废工位1（连续）
NGBox2	:INT:=6;		//	踢废工位2（单片）
BrushDustU	:INT:=7;		//	极片上表面毛刷除尘工位
WindDustU	:INT:=8;		//	极片上表面风刀除尘工位
BrushDustD	:INT:=9;		//	极片下表面毛刷除尘工位
WindDustD	:INT:=10;		//	极片下表面风刀除尘工位(除尘倒装皮带末位)
//DedustRevBelt     :INT;  //除尘倒装皮带末位
SubBelt1	:INT;		//	分段皮带1取料工位
SubBelt2	:INT;		//	分段皮带2取料工位
SubBelt3	:INT;		//	分段皮带3取料工位
END_STRUCT
END_TYPE

// ---- DUTs/33_M2/ST_IntervalData.TcDUT
TYPE ST_IntervalData ://极耳间距数据（裁断前）
STRUCT
	fTabIntervalM:					REAL;//倒角前CCD测出的极耳间距(相当于一个片宽)
	//fCen_RealWidthM_L:                REAL;//冲R角时左肩宽实时基准值
	//fCen_RealWidthM_R:                REAL;//冲R角时右肩宽实时基准值
	bTabInteFr_M:BOOL;//模具前，1=极耳间距前进方向(靠近裁切)肩宽NG
	bTabInteBe_M:BOOL;//模具前，1=极耳间距非前进方向(远离裁切)肩宽NG
	fTabIntervalC:                 REAL;//裁断前CCD测出的极耳间距(相当于一个片宽)
	//fCen_RealWidthC_L:                REAL;//裁断时左肩宽实时基准值
	//fCen_RealWidthC_R:                REAL;//裁断时右肩宽实时基准值
	bTabInteFr_C:BOOL;//模具前，1=极耳间距前进方向(靠近裁切)肩宽NG
	bTabInteBe_C:BOOL;//模具前，1=极耳间距非前进方向(远离裁切)肩宽NG	
	bBlueNG:                  BOOL;//1=蓝胶NG
	bLineScanNG:                  BOOL;//1=线扫NG
	bIntervalFail_M:                 BOOL;//true=极耳间距NG，倒角前CCD
	bIntervalFail_C:                 BOOL;//true=极耳间距NG，裁切前CCD
END_STRUCT
END_TYPE

// ---- DUTs/33_M2/ST_IntervalNo.TcDUT
TYPE ST_IntervalNo ://极耳间距工位（裁断前）
STRUCT
First	:INT:=1;		//	首工位（蓝胶检测位）1
Mould	:INT:=5;		//冲R角位  5
Cuter	:INT:=10;		//	裁切位    10
END_STRUCT
END_TYPE

// ---- DUTs/33_M2/ST_TabNo.TcDUT
TYPE ST_TabNo ://极耳工位（裁断前）
STRUCT
MouldPhoto	:INT:=1;		//首工位(R角CCD定位拍照位)   1
CuterPhoto	:INT:=6;		//首工位(裁切CCD定位拍照位)   6
LineScanNG	:INT:=3;			//线扫NG踢废位  3
END_STRUCT
END_TYPE

// ---- DUTs/34_M1/ST_CCDio.TcDUT
TYPE ST_CCDio :
STRUCT
   hmiChamferPhoto              :BOOL;       (***CCD冲R角定位拍照触发**)
   hmiCuterPhoto              :BOOL;       (***CCD裁切定位拍照触发**)
   hmiSizePhoto              :BOOL;       (***CCD尺寸检测拍照触发**)
   hmiXSPhoto:BOOL;//CCD线扫触发
   
   bCalibrationsDo_Cha   :BOOL;		(***CCD冲R角定位标定触发**)
   bCalibrationsDo_Cut   :BOOL;		(***CCD裁切定位标定触发**)
   bCalibrationsDo   :BOOL;		(***CCD冲R角&裁切定位标定同时触发**)
   
   bDemRuning   :BOOL;		(***标定运行中**)
   
   bCalibrationsDone_Cha   :BOOL;		(***CCD冲R角定位标定完成**)   
   bCalibrationsDone_Cut   :BOOL;		(***CCD裁切定位标定完成**)   
   
   bCalibrationsFals_Cha   :BOOL;		(***CCD冲R角定位标定失败**)   
   bCalibrationsFals_Cut   :BOOL;		(***CCD裁切定位标定失败**)   
   
   boChamferPhoto              :BOOL;       (***CCD冲R角定位拍照触发**)
   boCuterPhoto              :BOOL;       (***CCD裁切定位拍照触发**)
   boSizePhoto              :BOOL;       (***CCD尺寸检测拍照触发**)
   boXSPhoto:BOOL;//CCD线扫触发
END_STRUCT
END_TYPE

// ---- DUTs/35_CCD/ST_CCDComCuter.TcDUT
TYPE ST_CCDComCuter :
STRUCT
	fTabWidth:REAL;  //裁切定位CCD结果(极耳间距)
	fTabXOffset:REAL;  //裁切定位CCD结果(极片行进方向偏移)
	fTabYOffset:REAL;  //裁切定位CCD结果(极片横幅方向偏移)
	fTabXOffsetDeg:REAL;  //裁切定位CCD结果(极片行进方向角度)
	iFinish:INT;  //裁切定位CCD结果指示(1=视野内抓到极耳任意一个边   ;   2=视野内存在极耳，但极耳两个边都抓不到   ;   3:视野内不存在极耳;  )	
END_STRUCT
END_TYPE

// ---- DUTs/35_CCD/ST_CCDComLineScan.TcDUT
TYPE ST_CCDComLineScan :
STRUCT
	//BLineScanNG_Down   :INT;       (***线扫缺陷NG信号***)
	//BLineScanNG_UP   :INT;      
	bLineScanNG:BOOL; (***线扫缺陷NG信号***)
    bLineScan_Warn   :BOOL;       (***线扫暂停警告***)
	bLineScan_Estop   :BOOL;       (***线扫报警***)
	iResult:INT;  //先扫反馈结果(   1=OK   2=黄标类型(不停机)  ;3=裂纹圆角类型   ;0=无效)
	iPoleNo:STRING(256);//线扫极片编号
	iResult_Down:INT; //下线扫NG类型；
	iResult_UP:INT;//上线扫NG类型；
	iResult_Start:BOOL;//线扫软启动	
	bSendMark:BOOL;//PLC_To_PC上位机的发送数据标志
	
	(*******************************************线扫IO控制*****************************************************)
	iResult_IO_UP:INT;//上线扫结果	30=OK	31=NG	33=无效
	iResult_IO_Down:INT;//下线扫结果	30=OK	31=NG	33=无效
	
END_STRUCT
END_TYPE

// ---- DUTs/35_CCD/ST_CCDComR_Mould.TcDUT
TYPE ST_CCDComR_Mould :
STRUCT
    fTabXOffset:REAL;  //冲R角定位CCD结果(极片行进方向偏移)
	fTabYOffset:REAL;  //冲R角定位CCD结果(极片横幅方向偏移)
	iFinish:INT;  //冲R角定位CCD结果指示(1=视野内抓到极耳任意一个边   ;   2=视野内存在极耳，但极耳两个边都抓不到   ;   3:视野内不存在极耳;   )
END_STRUCT
END_TYPE

// ---- DUTs/35_CCD/ST_CCDComSize.TcDUT
TYPE ST_CCDComSize :
STRUCT
	fPoleWidth:REAL;  //尺寸检测CCD结果(极片宽度)
	fPoleHeigh:REAL;  //尺寸检测CCD结果(极片高度)
	fTabWidth:REAL;  //尺寸检测CCD结果(极耳宽度)
	fTabHeigh:REAL;  //尺寸检测CCD结果(极耳高度)
	fTabSite   : REAL; // 极耳左，右边距(就是极耳位置，不分左右)
	fOffsetDeg:REAL; //尺寸检测CCD结果(极片裁切面角度偏移)
	
	RoundedSize1                                :        REAL        ;//        圆角尺寸1 纵深
	RoundedSize2                                :        REAL        ;//        圆角尺寸2纵深
	RoundedSize3                                :        REAL        ;//        圆角尺寸3纵深
	RoundedSize4                                :        REAL        ;//        圆角尺寸4纵深
	RoundedSize5                                :        REAL        ;//        圆角尺寸5 横深
	RoundedSize6                                :        REAL        ;//        圆角尺寸6横深
	RoundedSize7                                :        REAL        ;//        圆角尺寸7横深
	RoundedSize8                               :        REAL        ;//        圆角尺寸8横深
	
	PolePlateAngle1                                :        REAL        ;//        极片角度1  极片角度
	PolePlateAngle2                                :        REAL        ;//        极片角度2
	PolePlateAngle3                                :        REAL        ;//        极片角度3
	PolePlateAngle4                                :        REAL        ;//        极片角度4
	
	fPoleNGSizeNo:REAL;  //尺寸检测CCD结果(NG分类编号)
	iTabNGSizeNo:INT;  //尺寸检测CCD极耳抓边异常分类     1： OK  2: 极片抓边异常    3:极耳抓边异常     4：都抓边异常     5：极片或极耳角度异常    
	
	iPoleRAngleNG:INT;//尺寸检测CCD结果(R角NG)
	iFinish:INT;  //尺寸检测CCD结果指示(1=完成;2=NG;3=无片;0=无效)  SizeResults
	
	AppearanceResult:INT;// 极片外观判定结果   线扫NG、OK
	stPoleNo:	STRING(256);//极片编号  PC 发送给PLC 预留   区分正负极
	
END_STRUCT
END_TYPE

// ---- DUTs/38_交互/DToM_Process.TcDUT
TYPE DToM_Process ://叠片→模切  生产过程数据
STRUCT
	bAn_M1Done:BOOL;//1号叠台正极取料完成
	bAn_M2Done:BOOL;//2号叠台正极取料完成
	bAn_M3Done:BOOL;//3号叠台正极取料完成
	
	bAn_M1Safety:BOOL;//1号叠台正极安全(取料运行时:=FALSE)
	bAn_M2Safety:BOOL;//2号叠台正极安全(取料运行时:=FALSE)
	bAn_M3Safety:BOOL;//3号叠台正极安全(取料运行时:=FALSE)
	
	bCa_M1Done:BOOL;//1号叠台负极取料完成
	bCa_M2Done:BOOL;//2号叠台负极取料完成
	bCa_M3Done:BOOL;//3号叠台负极取料完成
	
	bCa_M1Safety:BOOL;//1号叠台负极安全(取料运行时:=FALSE)
	bCa_M2Safety:BOOL;//2号叠台负极安全(取料运行时:=FALSE)
	bCa_M3Safety:BOOL;//3号叠台负极安全(取料运行时:=FALSE)	
	
	
	bAn_M1LockReady:BOOL;//1号叠台正极锁定准备好
	bAn_M2LockReady:BOOL;//2号叠台正极锁定准备好
	bAn_M3LockReady:BOOL;//3号叠台正极锁定准备好
		
	bCa_M1LockReady:BOOL;//1号叠台负极锁定准备好
	bCa_M2LockReady:BOOL;//2号叠台负极锁定准备好
	bCa_M3LockReady:BOOL;//3号叠台负极锁定准备好

	bAn_M1JumpReady:BOOL;//1号叠台正极锁定 未准备好
	bAn_M2JumpReady:BOOL;//2号叠台正极锁定 未准备好
	bAn_M3JumpReady:BOOL;//3号叠台正极锁定 未准备好
		
	bCa_M1JumpReady:BOOL;//1号叠台负极锁定 未准备好
	bCa_M2JumpReady:BOOL;//2号叠台负极锁定 未准备好
	bCa_M3JumpReady:BOOL;//3号叠台负极锁定 未准备好	
	
	bAn_M1LockingCancel:BOOL;//叠台1锁定中取消
	bAn_M2LockingCancel:BOOL;//叠台2锁定中取消
	bAn_M3LockingCancel:BOOL;//叠台3锁定中取消
	
	bCa_M1LockingCancel:BOOL;//叠台1锁定中取消
	bCa_M2LockingCancel:BOOL;//叠台2锁定中取消
	bCa_M3LockingCancel:BOOL;//叠台3锁定中取消	
	
	bAn_M1PoleHave:BOOL;//叠台1正极取料位无片
	bAn_M2PoleHave:BOOL;//叠台2正极取料位无片
	bAn_M3PoleHave:BOOL;//叠台3正极取料位无片
	
	bCa_M1PoleHave:BOOL;//叠台1负极取料位无片
	bCa_M2PoleHave:BOOL;//叠台2负极取料位无片
	bCa_M3PoleHave:BOOL;//叠台3负极取料位无片
	

	
END_STRUCT
END_TYPE

// ---- DUTs/38_交互/DToM_System.TcDUT
TYPE DToM_System ://叠片→模切  系统数据
STRUCT
	bP2M1Enable:BOOL;//TRUE 1号叠片启用
	bP2M2Enable:BOOL;//TRUE 2号叠片启用
	bP2M3Enable:BOOL;//TRUE 3号叠片启用
	
	bP2Estop:BOOL;//TRUE 叠片急停
	bP2Start:BOOL;//TRUE 叠片启动
	bP2Runing:BOOL;//TRUE 叠片自动中
	
//清尾料
	bP2ClearDo:BOOL;//叠片开始清尾料   注：先发需求量，再发清尾料开始信号
	iAn1Ask:INT:=0;// 1号正极极片需求量
	iAn2Ask:INT:=0;// 2号正极极片需求量
	iAn3Ask:INT:=0;// 3号正极极片需求量
	iCa1Ask:INT:=0;// 1号负极极片需求量
	iCa2Ask:INT:=0;// 2号负极极片需求量
	iCa3Ask:INT:=0;// 3号负极极片需求量
	bP2ClearDone:BOOL;//叠片清尾料完成	

//光电信号传递
	bAnBelt1Have:BOOL;//正极分段皮带1有料感应
	bAnBelt2Have:BOOL;//正极分段皮带2有料感应
	bAnBelt3Have:BOOL;//正极分段皮带3有料感应
	bCaBelt1Have:BOOL;//负极分段皮带1有料感应
	bCaBelt2Have:BOOL;//负极分段皮带2有料感应
	bCaBelt3Have:BOOL;//负极分段皮带3有料感应


	P3SaveParDone      :BOOL;//p3保存参数完成
	P3ReadParDone     :BOOL;//p3读取参数完成
	
	fM1MainSetPos:REAL;//叠片1主轴指令位置
	fM2MainSetPos:REAL;//叠片2主轴指令位置
	fM3MainSetPos:REAL;//叠片3主轴指令位置
	
END_STRUCT
END_TYPE

// ---- DUTs/38_交互/MToD_Process.TcDUT
TYPE MToD_Process ://模切→叠片  生产过程数据
STRUCT
	bAn_M1Allow:BOOL;//允许1号叠台正极取料
	bAn_M2Allow:BOOL;//允许2号叠台正极取料
	bAn_M3Allow:BOOL;//允许3号叠台正极取料

	bAn_M1Allow2:BOOL;//允许1号叠台正极取料
	bAn_M2Allow2:BOOL;//允许2号叠台正极取料
	bAn_M3Allow2:BOOL;//允许3号叠台正极取料
	
	bCa_M1Allow:BOOL;//允许1号叠台负极取料
	bCa_M2Allow:BOOL;//允许2号叠台负极取料
	bCa_M3Allow:BOOL;//允许3号叠台负极取料	
	
	bCa_M1Allow2:BOOL;//允许1号叠台负极取料
	bCa_M2Allow2:BOOL;//允许2号叠台负极取料
	bCa_M3Allow2:BOOL;//允许3号叠台负极取料		
	
	bAn_M1Locking:BOOL;//叠台1锁定中
	bAn_M2Locking:BOOL;//叠台2锁定中
	bAn_M3Locking:BOOL;//叠台3锁定中
	
	bCa_M1Locking:BOOL;//叠台1锁定中
	bCa_M2Locking:BOOL;//叠台2锁定中
	bCa_M3Locking:BOOL;//叠台3锁定中
END_STRUCT
END_TYPE

// ---- DUTs/38_交互/MToD_System.TcDUT
TYPE MToD_System ://模切→叠片  系统数据
STRUCT
	bP1Estop:BOOL;//TRUE 模切急停
	bP1Start:BOOL;//TRUE 模切启动
	bP1Runing:BOOL;//TRUE 模切自动中
	iCarryPoleMode:INT:=3;//极片仅流至1.2.3工位
	p1state:INT;//模切状态1:自动中   2:自动-Ready  3:手动   4:急停    5：报警    6.自动-NoReady
	P1SaveParDone      :BOOL;//模切保存参数完成
	P1ReadParDone     :BOOL;//模切读取参数完成
//清尾料
	bP1ClearDo:BOOL;//模切开始清尾料   注：模切部分程序必须在叠片开始清尾料后，在进入清尾料流程
	bP1ClearDone:BOOL;//模切清尾料完成	注：必须叠台部分叠完所有极片立马给模切 叠片清尾料完成，最后模切反馈清尾料完成
END_STRUCT
END_TYPE

// ---- DUTs/38_交互/ST_P2InteractPart.TcDUT
TYPE ST_P2InteractPart ://交互_正负区分
STRUCT
//→叠台
	M1Allow:BOOL;//允许1号叠台取料
	M2Allow:BOOL;//允许2号叠台取料
	M3Allow:BOOL;//允许3号叠台取料

//→叠台
	M1Allow2:BOOL;//允许1号叠台取料
	M2Allow2:BOOL;//允许2号叠台取料
	M3Allow2:BOOL;//允许3号叠台取料
	
//叠台→	
	M1Done:BOOL;//1号叠台取料完成
	M2Done:BOOL;//2号叠台取料完成
	M3Done:BOOL;//3号叠台取料完成
	
	M1LockReady:BOOL;//1号叠台准备好取极片
	M2LockReady:BOOL;//2号叠台准备好取极片
	M3LockReady:BOOL;//3号叠台准备好取极片
	
	M1JumpReady:BOOL;//1号叠台跳过取极片	
	M2JumpReady:BOOL;//2号叠台跳过取极片	
	M3JumpReady:BOOL;//3号叠台跳过取极片	
	
	M1Safety:BOOL;//1号叠台安全(取料运行时:=FALSE)
	M2Safety:BOOL;//2号叠台安全(取料运行时:=FALSE)
	M3Safety:BOOL;//3号叠台安全(取料运行时:=FALSE)
	
	iM1Ask:INT:=0;// 1号叠台极片需求量
	iM2Ask:INT:=0;// 2号叠台极片需求量
	iM3Ask:INT:=0;// 3号叠台极片需求量
	
	M1PoleHave:BOOL;//叠台1取料位无片,,TRue触发上升沿清数据
	M2PoleHave:BOOL;//叠台2取料位无片,,TRue触发上升沿清数据
	M3PoleHave:BOOL;//叠台3取料位无片,,TRue触发上升沿清数据

	
END_STRUCT
END_TYPE

// ---- DUTs/38_交互/ST_P2InteractPub.TcDUT
TYPE ST_P2InteractPub ://交互_公共
STRUCT
//→叠台
	bP1Estop:BOOL;//TRUE 模切急停
	bP1Start:BOOL;//TRUE 模切启动
	bP1Runing:BOOL;//TRUE 模切自动中
	
	bP1ClearDo:BOOL;//模切开始清尾料   注：模切部分程序必须在叠片开始清尾料后，在进入清尾料流程
	bP1ClearDone:BOOL;//模切清尾料完成	注：必须叠台部分叠完所有极片立马给模切 叠片清尾料完成，最后模切反馈清尾料完成
	
//叠台→		
	P2M1Enable:BOOL;//TRUE 1号叠片启用
	P2M2Enable:BOOL;//TRUE 2号叠片启用
	P2M3Enable:BOOL;//TRUE 3号叠片启用
	
	bP2Estop:BOOL;//TRUE 叠片急停
	bP2Start:BOOL;//TRUE 叠片启动
	bP2Runing:BOOL;//TRUE 叠片自动中
	
	bP2ClearDo:BOOL;//叠片开始清尾料   注：先发需求量，再发清尾料开始信号
	bP2ClearDone:BOOL;//叠片清尾料完成	
END_STRUCT
END_TYPE

// ---- DUTs/39_记忆/ST_Meney_Type.TcDUT
TYPE ST_Meney_Type :
STRUCT
	
UnreelingTension			:	REAL	;//	放卷张力
SlicingSpeed				:	REAL	;//	切片速度
PolePlateLenth				:	REAL	;//	极片长度（走带方向）				
PolePlateAngle1				:	REAL	;//	极片角度1
PolePlateAngle2				:	REAL	;//	极片角度2
PolePlateAngle3				:	REAL	;//	极片角度3
PolePlateAngle4				:	REAL	;//	极片角度4
PolePlateWidth				:	REAL	;//	极片宽度
RoundedSize1				:	REAL	;//	圆角尺寸1
RoundedSize2				:	REAL	;//	圆角尺寸2
RoundedSize3				:	REAL	;//	圆角尺寸3
RoundedSize4				:	REAL	;//	圆角尺寸4
AppearanceResult			:	BOOL	;//	极片外观判定结果
EarMargin_L					:	REAL	;//	极耳左边距
EarMargin_R					:	REAL	;//	极耳右边距
RoundedPlaneBurr1			:	REAL	;//	圆角平面毛刺1
RoundedPlaneBurr2			:	REAL	;//	圆角平面毛刺2
RoundedPlaneBurr3			:	REAL	;//	圆角平面毛刺3
RoundedPlaneBurr4			:	REAL	;//	圆角平面毛刺4
RoundEndBurr1				:	REAL	;//	圆角端面毛刺1
RoundEndBurr2				:	REAL	;//	圆角端面毛刺2
RoundEndBurr3				:	REAL	;//	圆角端面毛刺3
RoundEndBurr4				:	REAL	;//	圆角端面毛刺4
PolePieceCuttingPlaneBurr1	:	REAL	;//	极片裁切平面毛刺1
PolePieceCuttingPlaneBurr2	:	REAL	;//	极片裁切平面毛刺2
EndFaceBurr1				:	REAL	;//	极片裁切端面毛刺1
EndFaceBurr2				:	REAL	;//	极片裁切端面毛刺2
CutOffPowderWidth			:	REAL	;//	极片裁切掉粉宽度
SizeResults					:	BOOL	;//	极片尺寸判定结果

END_STRUCT
END_TYPE

// ---- DUTs/MES/DTM_Mes1.TcDUT
TYPE DTM_Mes1 :	//XFP20240315
STRUCT
	uOther		:ARRAY[0..19] OF UINT;	//信号交互		
	bFuncEN     :ARRAY[0..10] OF BOOL; //功能开关状态
END_STRUCT
END_TYPE

// ---- DUTs/MES/MTD_Mes1.TcDUT
TYPE MTD_Mes1 :
STRUCT
	rExcelRate	:ARRAY[0..99] OF REAL;	//优报表real	
	uOther		:ARRAY[0..19] OF DINT;	//信号交互	
    bFuncEN     :ARRAY[0..20] OF BOOL;	//功能开关状态
	
END_STRUCT
END_TYPE

// ---- DUTs/指纹/ST_FingerprintKey.TcDUT
TYPE ST_FingerprintKey :
STRUCT
	MachineId		: 	STRING(49);//指纹器编号	
	UserId			:	STRING(49);//用户名	
	UserClassLevel	: 	STRING(49);//用户权限	
	Fid				: 	STRING(49);//本地文件id	
	MatchScore		:	STRING(49);//指纹匹配评分	
	Result			: 	STRING(49);//匹配结果	
	FileName		: 	STRING(49);//本地文件路径	
END_STRUCT
END_TYPE

// ---- DUTs/01_AxisCO_Ntrol/MC_AxisParameter.TcDUT


TYPE MC_AxisParameter : (
(* PLCopen specific parameters *) (* Index-Group 0x4000 + ID*)
   CommandedPosition := 1,           (* lreal *) (* taken from NcToPlc *)
   SWLimitPos,                       (* lreal *) (* IndexOffset= 16#0001_000E *)
   SWLimitNeg,                       (* lreal *) (* IndexOffset= 16#0001_000D *)
   EnableLimitPos,                   (* bool  *) (* IndexOffset= 16#0001_000C *)
   EnableLimitNeg,                   (* bool  *) (* IndexOffset= 16#0001_000B *)
   EnablePosLagMonitoring,           (* bool  *) (* IndexOffset= 16#0002_0010 *)
   MaxPositionLag,                   (* lreal *) (* IndexOffset= 16#0002_0012 *)
   MaxVelocitySystem,                (* lreal *) (* IndexOffset= 16#0000_0027 *)
   MaxVelocityAppl,                  (* lreal *) (* IndexOffset= 16#0000_0027 *)
   ActualVelocity,                   (* lreal *) (* taken from NcToPlc *)
   CommandedVelocity,                (* lreal *) (* taken from NcToPlc *)
   MaxAccelerationSystem,            (* lreal *) (* IndexOffset= 16#0000_0101 *)
   MaxAccelerationAppl,              (* lreal *) (* IndexOffset= 16#0000_0101 *)
   MaxDecelerationSystem,            (* lreal *) (* IndexOffset= 16#0000_0102 *)
   MaxDecelerationAppl,              (* lreal *) (* IndexOffset= 16#0000_0102 *)
   MaxJerkSystem,                    (* lreal *) (* IndexOffset= 16#0000_0103 *)
   MaxJerkAppl,                      (* lreal *) (* IndexOffset= 16#0000_0103 *)

(* Beckhoff specific parameters *) (* Index-Group 0x4000 + ID*)
   AxisId := 1000,                   (* lreal *) (* IndexOffset= 16#0000_0001 *)
   AxisVeloManSlow,                  (* lreal *) (* IndexOffset= 16#0000_0008 *)
   AxisVeloManFast,                  (* lreal *) (* IndexOffset= 16#0000_0009 *)
   AxisVeloMax,                      (* lreal *) (* IndexOffset= 16#0000_0027 *)
   AxisAcc,                          (* lreal *) (* IndexOffset= 16#0000_0101 *)
   AxisDec,                          (* lreal *) (* IndexOffset= 16#0000_0102 *)
   AxisJerk,                         (* lreal *) (* IndexOffset= 16#0000_0103 *)
   MaxJerk,                          (* lreal *) (* IndexOffset= 16#0000_0103 *)
   AxisMaxVelocity,                  (* lreal *) (* IndexOffset= 16#0000_0027 *)
   AxisRapidTraverseVelocity,        (* lreal *) (* IndexOffset= 16#0000_000A *)
   AxisManualVelocityFast,           (* lreal *) (* IndexOffset= 16#0000_0009 *)
   AxisManualVelocitySlow,           (* lreal *) (* IndexOffset= 16#0000_0008 *)
   AxisCalibrationVelocityForward,   (* lreal *) (* IndexOffset= 16#0000_0006 *)
   AxisCalibrationVelocityBackward,  (* lreal *) (* IndexOffset= 16#0000_0007 *)
   AxisJogIncrementForward,          (* lreal *) (* IndexOffset= 16#0000_0018 *)
   AxisJogIncrementBackward,         (* lreal *) (* IndexOffset= 16#0000_0019 *)
   AxisEnMinSoftPosLimit,            (* bool  *) (* IndexOffset= 16#0001_000B *)
   AxisMinSoftPosLimit,              (* lreal *) (* IndexOffset= 16#0001_000D *)
   AxisEnMaxSoftPosLimit,            (* bool  *) (* IndexOffset= 16#0001_000C *)
   AxisMaxSoftPosLimit,              (* lreal *) (* IndexOffset= 16#0001_000E *)
   AxisEnPositionLagMonitoring,      (* bool  *) (* IndexOffset= 16#0002_0010 *)
   AxisMaxPosLagValue,               (* lreal *) (* IndexOffset= 16#0002_0012 *)
   AxisMaxPosLagFilterTime,          (* lreal *) (* IndexOffset= 16#0002_0013 *)
   AxisEnPositionRangeMonitoring,    (* bool  *) (* IndexOffset= 16#0000_000F *)
   AxisPositionRangeWindow,          (* lreal *) (* IndexOffset= 16#0000_0010 *)
   AxisEnTargetPositionMonitoring,   (* bool  *) (* IndexOffset= 16#0000_0015 *)
   AxisTargetPositionWindow,         (* lreal *) (* IndexOffset= 16#0000_0016 *)
   AxisTargetPositionMonitoringTime, (* lreal *) (* IndexOffset= 16#0000_0017 *)
   AxisEnInTargetTimeout,            (* bool  *) (* IndexOffset= 16#0000_0029 *)
   AxisInTargetTimeout,              (* lreal *) (* IndexOffset= 16#0000_002A *)
   AxisEnMotionMonitoring,           (* bool  *) (* IndexOffset= 16#0000_0011 *)
   AxisMotionMonitoringWindow,       (* lreal *) (* IndexOffset= 16#0000_0028 *)
   AxisMotionMonitoringTime,         (* lreal *) (* IndexOffset= 16#0000_0012 *)
   AxisDelayTimeVeloPosition,        (* lreal *) (* IndexOffset= 16#0000_0104 *)
   AxisEnLoopingDistance,            (* bool  *) (* IndexOffset= 16#0000_0013 *)
   AxisLoopingDistance,              (* lreal *) (* IndexOffset= 16#0000_0014 *)
   AxisEnBacklashCompensation,       (* bool  *) (* IndexOffset= 16#0000_002B *)
   AxisBacklash,                     (* lreal *) (* IndexOffset= 16#0000_002C *)
   AxisEnDataPersistence,            (* bool  *) (* IndexOffset= 16#0000_0030 *)
   AxisRefVeloOnRefOutput,           (* lreal *) (* IndexOffset= 16#0003_0101 *)
   AxisOverrideType,                 (* lreal *) (* IndexOffset= 16#0000_0105 *)
   (* new since 4/2007 *)
   AxisEncoderScalingFactor,         (* lreal *) (* IndexOffset= 16#0001_0006 *)
   AxisEncoderOffset,                (* lreal *) (* IndexOffset= 16#0001_0007 *)
   AxisEncoderDirectionInverse,      (* bool  *) (* IndexOffset= 16#0001_0008 *)
   AxisEncoderMask,                  (* dword *) (* IndexOffset= 16#0001_0015 *)
   AxisEncoderModuloValue,           (* lreal *) (* IndexOffset= 16#0001_0009 *)
   AxisModuloToleranceWindow,        (* lreal *) (* IndexOffset= 16#0001_001B *)
   AxisEnablePosCorrection,          (* bool  *) (* IndexOffset= 16#0001_0016 *)
   AxisPosCorrectionFilterTime,      (* lreal *) (* IndexOffset= 16#0001_0017 *)
   (* new since 1/2010 *)
   AxisUnitInterpretation,           (* lreal *) (* IndexOffset= 16#0000_0026 *)
   AxisMotorDirectionInverse,        (* bool  *) (* IndexOffset= 16#0003_0006 *)
   (* new since 1/2011 *)
   AxisCycleTime,                    (* lreal *) (* IndexOffset= 16#0000_0004 *)
   (* new since 5/2011 *)
   AxisFastStopSignalType,           (* dword *) (* IndexOffset= 16#0000_001E *)
   AxisFastAcc,                      (* lreal *) (* IndexOffset= 16#0000_010A *)
   AxisFastDec,                      (* lreal *) (* IndexOffset= 16#0000_010B *)
   AxisFastJerk,                     (* lreal *) (* IndexOffset= 16#0000_010C *)

(* Beckhoff specific axis status information - READ ONLY *) (* Index-Group 0x4100 + ID*)
   AxisTargetPosition := 2000,       (* lreal *) (* IndexOffset= 16#0000_0013 *)
   AxisRemainingTimeToGo,            (* lreal *) (* IndexOffset= 16#0000_0014 *)
   AxisRemainingDistanceToGo,        (* lreal *) (* IndexOffset= 16#0000_0022, 16#0000_0042 *)

(* Beckhoff specific axis functions *)
   (* read/write gear ratio of a slave *)
   AxisGearRatio := 3000,            (* lreal *) (* read: IndexGroup=0x4100+ID, IdxOffset=16#0000_0022, *)
                   (* write:IndexGroup=0x4200+ID, IdxOffset=16#0000_0042 *) 

(* Beckhoff specific other parameters *)
   (* new since 1/2011 *)
   NcSafCycleTime := 4000,           (* lreal *) (* IndexOffset= 16#0000_0010 *)
   NcSvbCycleTime                    (* lreal *) (* IndexOffset= 16#0000_0012 *)
);
END_TYPE

// ---- DUTs/01_AxisCO_Ntrol/ST_SetpMotor.TcDUT
TYPE ST_SetpMotor :
STRUCT
	bJog_Up			:BOOL;		//手动上升
	bJog_Down			:BOOL;	 //手动下降
	bHome			:BOOL;	 //回原点启动
	bGoWorkPos			:BOOL;	 //定位至工作位(上升)
	bLeaveWorkPos			:BOOL;	 //定位脱离工作位(下降)
	HomeDone    :BOOL;  //回原点完成
	WorkPosDone :BOOL;//定位完成
	
	
	
	biSensor  :BOOL;   //高度对射光电
	biUpSensor  :BOOL;//电机上限
	//biRefSensor  :BOOL;   //电机原点
	biBoxSensor  :BOOL;   //料盒到位感应
	biDownSensor  :BOOL;  //电机下限
	
	bError:ARRAY[1..3]  OF BOOL; 
	
	bo_Up			:BOOL;		//电机上升
	bo_Down			:BOOL;//电机下降

	bPoleFull: BOOL;  //极片料满

END_STRUCT
END_TYPE

// ---- DUTs/08_IO/ST_MoQieSenser.TcDUT
TYPE ST_MoQieSenser ://传感器
STRUCT
	biFlgBlue              :BOOL;       (***极片接带检测1***)
	biCuterStopUp                :BOOL;       (***裁切切刀堵料检测***)
	biSafetyCurtain_M                :BOOL;       (***模具安全光幕**)
	biSafetyCurtain_C                :BOOL;       (***裁切安全光幕**)
	biWasteBox               :BOOL;       (***废料收集箱高度感应**)
	biTabHave               :BOOL;       (***极耳有无感应**)
	
	biSubBelt1Have                    :BOOL;       (***分段皮带1有料感应**)
	biSubBelt2Have                    :BOOL;       (***分段皮带2有料感应**)
	biSubBelt3Have                    :BOOL;       (***分段皮带3有料感应**)   
	
	biDoor                       :ARRAY [1..5] OF BOOL;  (***门禁**)		
	
	aiPoleTensionFr               :REAL;       (***辅驱前极片张力检测***)
	aiPoleTensionBe               :REAL;       (***辅驱后极片张力检测***)	
	
	aiMouldRectifyFr              :REAL;       (***倒角深度前纠偏检测**)
	aiMouldRectifyBe               :REAL;      (***倒角深度后纠偏检测**)	
	
	biCutPoleHave					:BOOL;//裁切后极片有无检测
	bKick:BOOL;//踢废工位是否有料检测；
	bYellowCheck_C:BOOL;//踢废前黄标检测感应器
	bYellowCheck_R1:BOOL;//倒角前黄标检测感应器上
	bYellowCheck_R2:BOOL;//倒角前黄标检测感应器下
	bPoleCheck_R:BOOL;//倒角前极耳检测感应器
	aThrow:BOOL;  
	NGBoxFull:BOOL;//NG料盒料满信号
	
(***************************************************线扫20240219***********************************************************************)
	bLineScanResult1_UP:BOOL;//上线扫结果NG
	bLineScanResult2_UP:BOOL;//上线扫结果OK
	bLineScanResult1_Down: BOOL;//下线扫结果NG
	bLineScanResult2_Down:BOOL;//下线扫结果OK
	
	NGboxsensor 	:BOOL;		//模切NG料盒抛料对射感应		
    MouldInsensor       :BOOL;		//R角模具到位感应
    CuterInsensor       :BOOL;		//裁切切刀到位感应
	bFourYellowUP		:BOOL;		//四连标上
	bFourYellowDown:BOOL;		//四连标下
END_STRUCT
END_TYPE

// ---- DUTs/08_IO/ST_MoQieButton.TcDUT
TYPE ST_MoQieButton :// 按钮
STRUCT
    PoleBoxBit1                       :BOOL;    (**极片放卷按钮BIT1**)
    PoleBoxBit2                       :BOOL;    (**极片放卷按钮BIT2**)
    PoleBoxBit3                       :BOOL;    (**极片放卷按钮BIT3**)
    PoleBoxBit4                       :BOOL;    (**极片放卷按钮BIT4**)
    PoleBoxStart                        :BOOL;    (**极片放卷启动按钮*)
    PoleBoxEStop                      :BOOL;    (**极片放卷紧急停止*)
	
	CoderRollPress                      :BOOL; (**编码器辊压辊按钮*)
	
    DriverPress_Aux                        :BOOL;   (**辅驱压辊旋钮**)
	DriverJogFw_Aux                       :BOOL;    (**辅助驱辊正向点动*)
	DriverJogBw_Aux                        :BOOL;   (**辅助驱辊反向点动**)
	
	DriverPressDDR                      :BOOL; (**主驱动压辊按钮*)
	
    NGBoxStart                         :BOOL;  (**NG料盒面板确认按钮**)
    NGBoxEStop                       :BOOL;  (**NG料盒面板急停按钮**)
    NGBoxMotor_JogUp                       :BOOL;  (**NG料盒面板排杆电机手动上升**)
    NGBoxMotor_JogDown                      :BOOL;  (**NG料盒面板排杆电机手动下降**)
	
    PoleBrushDustPush_U                        :BOOL;  (**正极上表面毛刷除尘升降气缸按钮*)
	PoleWindDustPush_U                        :BOOL;  (**正极上表面风刀除尘升降气缸按钮*)
	PoleBrushDustPush_D                        :BOOL;  (**正极下表面毛刷除尘升降气缸按钮*)
	PoleWindDustPush_D                        :BOOL;  (**正极下表面风刀除尘升降气缸按钮*)
(**外罩急停*)
  	EncloserEstop                      :ARRAY [1..3] OF BOOL;    (**外罩紧急停止*)
	
(**按钮指示灯*)
    PoleBoxStartLight                         :BOOL;    (**极片放卷启动按钮指示灯*)
    DriverPressDDRLight                       :BOOL; (**主驱动压辊按钮指示灯*)
	CoderRollPressLight                      :BOOL; (**编码器辊压辊按钮指示灯*)
	
    NGBoxStartLight                         :BOOL;  (**NG料盒面板确认按钮指示灯**)
    NGBoxMotor_JogUpLight                   :BOOL;  (**NG料盒面板排杆电机手动上升按钮指示灯**)
    NGBoxMotor_JogDownLight               :BOOL;  (**NG料盒面板排杆电机手动下降按钮指示灯**)
	
    PoleBrushDustPush_ULight                       :BOOL;  (**正极上表面毛刷除尘升降气缸按钮指示灯*)
	PoleWindDustPush_ULight                       :BOOL;  (**正极上表面风刀除尘升降气缸按钮指示灯*)
	PoleBrushDustPush_DLight                        :BOOL;  (**正极下表面毛刷除尘升降气缸按钮指示灯*)
	PoleWindDustPush_DLight                        :BOOL;  (**正极下表面风刀除尘升降气缸按钮指示灯*)
	
(**按钮指示灯*)
	iPoleBoxCode:       							INT;(*极片放卷按钮盒编码开关指示*)	

END_STRUCT
END_TYPE

// ---- DUTs/07_Name/ST_AxisName.TcDUT
TYPE ST_AxisName :   //轴名称
STRUCT
UnWind_L	:INT;//模切左放卷
UnWind_R	:INT;//模切右放卷
PoleTension	:INT;//模切前摆杆张力
DriverAux	:INT;//模切辅助驱动
BuffeLine	:INT;//模切极片缓存1:初始位 2：正极限位 3：负极限位
Mould	:INT;//倒角模具
MouldRectify_X	:INT;//模具纠偏X轴(肩宽补偿)
MouldRectify_Y	:INT;//模具纠偏Y轴(切刀深度)
DriverDDR	:INT;//模切主驱动
Cuter	:INT;//裁切切刀
CuterDegRectify	:INT;//裁切角度纠偏
CuterBelt	:INT;//裁切输送皮带
CuterBeltChange	:INT;//裁切输送带换型
CCDPressPush	:INT;//尺寸CCD压片升降
NGPushReverseBelt	:INT;//踢废倒装皮带
NGPush1	:INT;//踢连续废料
NGPush2	:INT;//踢单张废料
DedustBelt	:INT;//上表面除尘皮带
DedustReverseBelt	:INT;//下表面除尘倒装皮带
SubBelt1	:INT;//送料分段皮带1
SubBelt2	:INT;//送料分段皮带2
SubBelt3	:INT;//送料分段皮带3
Ready1	:INT;//备用1
Ready2	:INT;//备用2
END_STRUCT
END_TYPE

// ---- DUTs/07_Name/ST_RecName.TcDUT
TYPE ST_RecName :   //  纠偏名称
STRUCT
      PoleWind          :INT; (***极片放卷纠偏*)
      PoleProcess      :INT; (***极片行进纠偏*)
END_STRUCT
END_TYPE

// ---- DUTs/07_Name/ST_ElectValveName.TcDUT
TYPE ST_ElectValveName :   //阀名称
STRUCT
ConnectDustVacuo	:INT;	//	极片接带平台除尘真空
LineSceneDustBlow	:INT;	//	线扫相机镜头除尘吹气
LineSceneDustVacuo	:INT;	//	线扫相机镜头除尘真空
AreaArrayDustBlow	:INT;	//	模切面阵相机镜头除尘吹气
MouldUpBlow	:INT;	//	模具上模吹气
MouldDownVacuo	:INT;	//	模具下模真空
MouldDownAir	:INT;	//	模具下模破真空
NGPushInsideAir	:INT;	//	NG踢废腔室破真空
NGPushInsideVacuo	:INT;	//	NG踢废腔室真空
BrushDustVacuo_U	:INT;	//	上表面毛刷除尘真空
WindDustBlow_U	:INT;	//	上表面风刀除尘吹气
WindDustVacuo_U	:INT;	//	上表面风刀除尘真空
BrushDustVacuo_D	:INT;	//	下表面毛刷除尘真空
WindDustBlow_D	:INT;	//	下表面风刀除尘吹气
WindDustVacuo_D	:INT;	//	下表面风刀除尘真空
RJ_Blow			:INT;//R角吹气
RJDustBlow  :INT;//R角风刀吹气
END_STRUCT
END_TYPE

// ---- DUTs/32_系统/IModeEN.TcDUT
TYPE IModeEN ://功能屏蔽
STRUCT
	bFounctionClose:ARRAY[1..20] OF BOOL;//1: 门襟屏蔽 2:风机报警屏蔽
	bDoorEN:BOOL:=TRUE;//TRUE  门襟屏蔽
	bBuzzerEN:BOOL:=TRUE;//TRUE 蜂鸣器屏蔽
    //bShortTestEN:BOOL;//TRUE 短路测试屏蔽
    //bCodeEN:BOOL;//TRUE 扫码屏蔽
    bCcdTcpEN:BOOL:=TRUE;  //TRUE ccd通讯屏蔽
	iModeRun:INT;//运行模式  1:仅正运行   2:仅负运行  0:正负运行   
	bNG2PushEN:BOOL:=TRUE;//TRUE NG踢单张料屏蔽
	iNGPole:INT:=10;//NG多少片后，料盒下降→上升一次
	iNGcyCout:INT:=3;//NG打料多少片后，归正气缸动作一次
	iCarryPoleMode:INT:=3;//极片流至1.2.3号工位。
	
	iNgSizeEN:INT:=3;//尺寸检测连续NG多少片后，报警
	iNgScaneEN:INT:=3;//线扫检测连续NG多少片后，报警
	
	
	bCuterOffsetEN:BOOL;//TRUE  裁切补偿（行进方向）屏蔽
	bMouldXOffsetEN:BOOL;//TRUE  模具X方向补偿（行进方向）屏蔽
	bMouldYRecEN:BOOL;//TRUE  模具Y方向纠偏（非行进方向）屏蔽
	bDegreeRecEN:BOOL;//TRUE  裁切角度纠偏屏蔽
	bNG1PushEN:BOOL;//TRUE NG踢连续料屏蔽

	bP2PartEN:BOOL:=TRUE;//TRUE 与叠片部分屏蔽
	bLineScanCCDEN:BOOL;//TRUE  线扫CCD屏蔽	
	bChamferCCDEN:BOOL;//TRUE  冲R角定位CCD屏蔽	
	bCuterCCDEN:BOOL;//TRUE  裁切定位CCD屏蔽
	bSizeCCDEN:BOOL;//TRUE  尺寸检测CCD屏蔽
	bFlgBlueEN:BOOL;//TRUE  蓝胶检测屏蔽
	bEmptyRunEN:BOOL;//TRUE 空跑模式
	bDedustEN:BOOL;//TRUE 除尘屏蔽
	bPoleCheckEN:BOOL;//堵料感应器屏蔽
	PartNumberOff    				: BOOL;   //物料校验功能屏蔽
	bTabWidtNGoff:BOOL;//连续极耳NG来料不良功能屏蔽
	bMouldXclosureEN:BOOL;//TRUE  模具X方向闭环（行进方向）屏蔽
	bMouldYclosureEN:BOOL;//TRUE  模具Y方向闭环（行进方向）屏蔽
END_STRUCT
END_TYPE

// ---- DUTs/32_系统/IRecipe.TcDUT
TYPE IRecipe :
STRUCT
	bCreate:BOOL;
	bSave:BOOL;
	bLoad:BOOL;

     
END_STRUCT
END_TYPE

// ---- DUTs/32_系统/ST_SysCmd.TcDUT
TYPE ST_SysCmd :
STRUCT

(*主页面指令*)
	bInit							:BOOL;	(*初始化*)

	bShutDownPc					:BOOL;	(*关机，程序做延迟*)
	bRebootPc						:BOOL;	(*重启PC*)
	bSaveData						:BOOL;	(*保存所有参数*)
    bReadData						:BOOL;	(*读取所有参数*)


END_STRUCT
END_TYPE

// ---- DUTs/32_系统/ST_SystemPublic.TcDUT
TYPE ST_SystemPublic ://系统功能块UDT
STRUCT

(***btn***)
	 btnStart                      :BOOL;  //启动按钮汇总
     btnStop                      :BOOL;  //停止按钮汇总
	 btnReset                     :BOOL;  //复位按钮汇总
     btnAuto                      :BOOL;//true=自动；false=手动 按钮汇总
	 btnEstop                    :BOOL;//急停按钮汇总	 

(***IO***)
   boRedLight                     :BOOL;           (***三色红灯***)
   boYellowLight                     :BOOL;           (***三色黄灯***)
   boGreenLight                      :BOOL;           (***三色绿灯***)
   boBuzzer							:BOOL;(***蜂鸣器***)
   
(***HMI*) 
	 iModehmi                  :INT;  //设备状态  1:自动中   2:自动-Ready  3:手动   4:急停    5：报警    6.自动-NoReady
	 hmiStart                    :BOOL;  
     hmiStop                    :BOOL;   
	 hmiReset                   :BOOL;  
     hmiAutoSwitch           :BOOL;
     hmiAuto                    :BOOL;
     hmiManul                  :BOOL;	 
	 hmiEstop                   :BOOL;
     hmiTest                     :BOOL;
	 //hmiGoHomeAll			:BOOL;
	 //hmiAllHomed			:BOOL;
(**Status**)
	 FlgAuto                     :BOOL;       //自动中标志位 硬件状态
	 FlgManua                  :BOOL;      //手动状态硬件状态
     iMode                       :INT;  //整机状态  1:自动中   2:暂停  3:手动   4:急停   
	   
	
     Autoing                     :BOOL;   //自动运行中
	 Manuling                   :BOOL;  //手动运行中
	 Stoping                     :BOOL;   //停止中
	 Alarming                   :BOOL;   //报警中
	 bErrorStop                :BOOL;//报警停机

     bAutoCondition         :BOOL;
     bStopFinished            :BOOL;
	 
	 bReset                      :BOOL; 
(*(***INIT***)
    bAnInit                        :BOOL;
    bCaInit                        :BOOL;
//    bP3Init                        :BOOL;
//    bP4Init                        :BOOL;
    bAnInitDone                :BOOL;
    bCaInitDone                :BOOL;
//    bP3InitDone                :BOOL;
//    bP4InitDone                :BOOL;
*)
	bInit							:BOOL;
    bInitDone                    :BOOL;
(**监控**)
	
   bwindow	          :BOOL;  // 弹窗         
   bAnccdstate        :BOOL;  //状态
   bCaccdstate        :BOOL;  //状态
END_STRUCT
END_TYPE

// ---- DUTs/06_Interface/IData.TcDUT
TYPE IData :
STRUCT
	strBetryName:STRING;//CCD给电芯名称 
	bNGOverHang :BOOL;  //
	bHaveBetry :BOOL;   //当前工位是否有电芯
    
	
	bNGShort:BOOL;  //短路NG
	strShortData:STRING; //短路测试数据
	
	strCode:STRING;//二维码
    bNGCode:BOOL;   //二维码NG
	
	strHotPress:STRING;//热压参数
END_STRUCT
END_TYPE

// ---- DUTs/06_Interface/IM2Glue.TcDUT
TYPE IM2Glue :  //备胶方法st
STRUCT
    Start1:BOOL;   //备胶启动
	Done1:BOOL;   //备胶完成
	bActioning:BOOL;//备胶动作中	
	bAction2ing:BOOL;//贴胶动作中	

	Start2:BOOL;   //贴胶启
	iTagetPos : INT;  //贴胶位置
    Done2:BOOL;  //贴胶动作完成
	

	Reset:BOOL;  //复位
	AutoRuning:BOOL;  //运行中信号

END_STRUCT
END_TYPE

// ---- DUTs/36_ShortTest/CMD.TcDUT
TYPE CMD :
STRUCT
	RST :                   STRING:='*RST';     // 1 仪器初始化
    Start :                 STRING:=':STARt';// 2 测试开始
    Stop :                  STRING:=':STOP';// 3  测试停止
    State_Check :           STRING:=':STATe?';// 4 测试状态查询 0：停止中  1：测试中   2：放电中
	
    Measure_Check :         STRING:=':MEASure?';// 5  测量值查询
    Measure_Check2 :        STRING:=':MEASure:RESult?';// 6  测量值，判定结果查询  //1:OFF 2:NOcomp 3:DELAY 4:PASS 5:UFAIL 6:LFAIL 7:ULFA
    Measure_Clear :         STRING:=':MEASure:CLEar';// 7  测量值，判定结果清除
	
    Voltage :               STRING:=':VOLTage';// 8  测试电压设置
    Voltage_Check :         STRING:=':VOLTage?';// 9  测试电压查询 
    Voltage_Monitor :       STRING:=':MEASure:MONItor?';// 10  电压值监视
	
    Mohm_Range :            STRING:=':MOHM:RANGe';// 11  电阻量程设置(2M/20M/200M/2000M/4000M/AUTO)  
    Mohm_Range_Check :      STRING:=':MOHM:RANGe?';// 12  电阻量程查询
	
    Speed :                 STRING:=':SPEed';// 13 测量速度设置(FAST/SLOW)
    Speed_Check :           STRING:=':SPEed?';// 14 测量速度查询
	
    Timer :                 STRING:=':TIMer';// 15  测试时间设置
    Timer_Check :           STRING:=':TIMer?';// 16  测试时间查询
    Delay :                 STRING:=':DELay';// 17  响应时间设置(0为自动)
    Delay_Check :           STRING:=':DELay?';// 18  响应时间查询(0为自动)
	
    ComparatorLimit :       STRING:=':COMParator:LIMit';// 19  比较器上下限值设置（上限,下限）
    ComparatorLimit_Check : STRING:=':COMParator:LIMit?';// 20  比较器上下限值查询
    ComparatorMode :        STRING:=':COMParator:MODE';// 21  测试模式设置（CONTinue/PASSstop/FAILstop/SEQuence）  
    ComparatorMode_Check :  STRING:=':COMParator:MODE?';// 22 测试模式查询（CONTINUE/PASSSTOP/FAILSTOP/SEQUENCE）
    ComparatorBeeper :      STRING:=':COMParator:BEEPer';// 23  判定蜂鸣器设置(PASS/FAIL/OFF/END)
    ComparatorBeeper_Check :STRING:=':COMParator:BEEPer?';// 24  判定蜂鸣器查询(PASS/FAIL/OFF/END)
	
    Contact :               STRING:=':CONTactcheck';//  25  接触检查功能设置(ON/OFF)	
	Contact_Check :         STRING:=':CONTactcheck?';// 26  接触检查功能查询(ON/OFF)
    Contact_Result :        STRING:=':CONTactcheck:RESult?';// 27  接触检查结果查询(NOCHK/PASS/HFAIL/LFAIL/HLFAIL)
	
    Short :                 STRING:=':SHORtcheck';// 28  短路检查功能设置(ON/OFF)	
    Short_Check :           STRING:=':SHORtcheck?';// 29  短路检查功能查询 
    ShortTime :             STRING:=':SHORtcheck:TIME';// 30 短路检查时间设置(0:自动)
    ShortTime_Check :       STRING:=':SHORtcheck:TIME?';// 31  短路检查时间查询
    Short_Result :          STRING:=':SHORtcheck:RESult?';// 32  短路检查结果查询（NOCHK/PASS/FAIL）
	
    KeyBeeper :             STRING:=':KEY:BEEPer';// 33  按键输入蜂鸣器音设置(ON/OFF)	
    KeyBeeper_Check :       STRING:=':KEY:BEEPer?';// 34  按键输入蜂鸣器音查询
   
END_STRUCT
END_TYPE

// ---- DUTs/36_ShortTest/IShortTest.TcDUT
TYPE IShortTest : 
STRUCT
	bStart :BOOL; //
	bDone  :BOOL; //

   iResult:INT; // 1 OK  2 NG
    
   ErrorID :INT;
   
	

END_STRUCT
END_TYPE

// ---- DUTs/36_ShortTest/ShortDataShow.TcDUT
TYPE ShortDataShow :
STRUCT
	strState:STRING;         //0：停止中  1：测试中   2：放电中
    strResult:STRING;  //启动测试后返回结果   综合结果
	
	strMeasure :STRING;     //测量电阻值
	strMeasureState :STRING;     //1:OFF 2:NOcomp 3:DELAY 4:PASS 5:UFAIL 6:LFAIL 7:ULFAIL

	strVoltageSetValue:STRING;  //电压设定值查询
    strVoltageMonitor:STRING; //电压值监视
	
	strMohmRangeValue:STRING;//(1:2M/2:20M/3:200M/4:2000M/5:4000M/6:AUTO) 
    
	strSpeedValue:STRING ;//测量速度查询(FAST/SLOW)
	
	strTimerValue :STRING;  //测试时间查询
	strDelayValue :STRING;  //响应时间查询(0自动）
	
	strComparatorLimitSet :STRING;  //比较器上限 下限值
	strComparatorModeValue: STRING ;// 21  测试模式查询（CONTinue/PASSstop/FAILstop/SEQuence）
	strComparatorBeeperValue:    STRING;//23  判定蜂鸣器查询(PASS/FAIL/OFF/END)
	
	strContactValue :STRING;//  25  接触检查功能查询(ON/OFF)
	strContactResult :STRING;//  27  接触检查结果查询(NOCHK/PASS/HFAIL/LFAIL/HLFAIL)
	
	strShortValue:STRING;// 28  短路检查功能查询(ON/OFF)
	strShortTimeValue:  STRING;// 30 短路检查时间查询(0:自动)
	strShortResult:STRING;// 32  短路检查结果查询（NOCHK/PASS/FAIL）
	
	strKeyBeeperValue:STRING;  // 33  按键输入蜂鸣器音查询(ON/OFF)	

END_STRUCT
END_TYPE

// ---- DUTs/36_ShortTest/ShortPar.TcDUT
TYPE ShortPar :
STRUCT
	fVoltageSet: REAL;  //电压设定值

	StrMohmRangeSet:STRING; //电阻量程设置(1:2M/2:20M/3:200M/4:2000M/5:4000M/6:AUTO) 

    StrSpeedSet:STRING ;//测量速度设置(FAST/SLOW)
    
    fTimerSet:    REAL; //测试时间设置
    fDelaySet:   REAL; //响应时间设定
     
	fComparatorUpLimitSet :REAL;  //比较器上限设定
	fComparatorDownLimitSet :REAL;//比较器下限设定	
    strComparatorModeSet: STRING ;// 21  测试模式设置（CONTinue/PASSstop/FAILstop/SEQuence）
	
	strComparatorBeeperSet:    STRING;//23  判定蜂鸣器设置(PASS/FAIL/OFF/END)
	
	strContactSet :STRING;//  25  接触检查功能设置(ON/OFF)	

	strShortSet:STRING;// 28  短路检查功能设置(ON/OFF)
	
	fShortTimeSet:  REAL;// 30 短路检查时间设置(0:自动)
	
	
	strKeyBeeperSet:STRING;  // 33  按键输入蜂鸣器音设置(ON/OFF)	
	
	
END_STRUCT
END_TYPE

// ---- DUTs/37_Code/ICode.TcDUT
TYPE ICode : 
STRUCT
	bComOpen:BOOL;  //扫码Tcp 开
    bComClose:BOOL;  //扫码Tcp 关

	bLON :BOOL; //  扫码开
	bLOFF :BOOL; //扫码关
	bDone  :BOOL; //扫码完成
    bError :BOOL;//扫码故障	
    strCode:STRING;//条码结果
    bCodeConError:BOOL;
END_STRUCT
END_TYPE

// ---- DUTs/35_CCD/ST_CCDCom.TcDUT
TYPE ST_CCDCom : 
STRUCT
	bLineHeart :BOOL;  //模切线扫相机部分软件心跳
	bAreaHeart:BOOL;//模切面阵相机部分软件心跳
	iDemResult_Cut:INT;//裁切定位标定结果指示(1=OK;2=NG;0=无效)
	iDemResult_Cha:INT;//冲R角定位标定结果指示(1=OK;2=NG;0=无效)
	
	iDemCount:INT;//标定拍照计数
	fDemLength:REAL:=20;//标定长度
	
	Scan:ST_CCDComLineScan;//线扫工位
	Chamfer:ST_CCDComR_Mould;//倒角前极耳定位工位
	Cuter:ST_CCDComCuter;//裁切前极耳定位工位
	Size:ST_CCDComSize;//裁切后尺寸检测工位
	
	
	iLineScanPhotoCount:   DINT;     
	iLineScanReceiveResultCount_UP:     DINT;
	iLineScanReceiveResultCount_Down:   DINT;
	bLineScanPhotoCountClear  :BOOL;
	
END_STRUCT
END_TYPE

// ---- DUTs/35_CCD/STCcdData.TcDUT
TYPE STCcdData :
STRUCT
	iorder:DINT;  //功能码  2  3   4    
	strCode:STRING   ;//二维码
	strShortData: STRING; //短路测试数据 128
	strBetryName: STRING;//文件名
	strHotPress: STRING;//热压参数
END_STRUCT
END_TYPE

// ---- DUTs/35_CCD/STCcdDataSend.TcDUT
TYPE STCcdDataSend :
STRUCT
	iHead :DINT:=32767;
	iorder:DINT:=2;
	strCode:ARRAY[0..63] OF   BYTE    ;//二维码
	strShortData: ARRAY[0..127] OF BYTE; //短路测试数据 128
	strBetryName: ARRAY[0..31] OF BYTE;//文件名
	strHotPress: ARRAY[0..63] OF BYTE;//热压参数
    iEnd :DINT:=65535;
END_STRUCT
END_TYPE

// ---- DUTs/34_M1/ST_Rectify.TcDUT
TYPE ST_Rectify :   //纠偏控制
STRUCT
(********参数**************)	

	bReset            :BOOL;     // 纠偏复位  
	bEnable		:BOOL;	(*开启自动纠偏*)
	fSensorActValue			:REAL; //实际位置
	
	bReady              :BOOL;  //纠偏准备号
	bAutoRunning		:BOOL;	(*纠偏自动运行中*)
	Error		:BOOL;            //纠偏错误
    ErrID:	 STRING;     //纠偏错误代码
	
END_STRUCT
END_TYPE

// ---- DUTs/31_其他辅助/File_com_typ.TcDUT
TYPE File_com_typ :(*xml内部用*)
STRUCT
	FileName_save: 		T_MaxString	 := 'test.xml';		(* File name would be saved setting by the HMI用来保存的文件名称 *)
	FileName_active: 	T_MaxString	 := 'test.xml';		(* File name activated now to be loaded 用来读取的文件目标文件名*)
	Device: 			T_MaxString  := '\Hard Disk\';		(* Device: C:\ or USB    or ce   \Hard Disk\*)
	DeviceNum:		INT:=3;							(* 1= C:\ or 2=USB    or 3= ce   \Hard Disk\*)
	Var_Name: 			ARRAY [0..19] OF T_MaxString;	(* Variable name which need to be loaded or saved *)
	Dir_change:			BOOL;							(* Command for change the directory	*)
	File_load:			BOOL;							(* Command for load the exiting file	*)
	File_save:			BOOL;							(* Command for save the file	*)
	File_del:			BOOL;							(* Command for delete the exiting file	*)
	File_copy:			BOOL;							(* Command for copy the exiting file between the C:\ and USB *)
	Err_ack:			BOOL;							(* Command for acklonege the error	*)
	bBusy:				BOOL;							(* State for the FB running	*)
	ErrorID:			UDINT;							(* Error ID from the FB *)
END_STRUCT
END_TYPE

// ---- DUTs/31_其他辅助/ST_DATA_NEED_BE_PERSIS.TcDUT
TYPE ST_DATA_NEED_BE_PERSIS :(*需要断电保持的参数*)(*中间变量，只用在判断用*)
STRUCT

	strSetLevelPassword: 	ARRAY [0..3] OF STRING(80) := ['0','1','2','3'];
	strInputReceipeName: 	STRING(80);
	strCurrentReceipeName: 	STRING(80);

END_STRUCT
END_TYPE

// ---- GVLs/GVL_Par.TcGVL
VAR_GLOBAL    //参数
         
	         

END_VAR




VAR_GLOBAL PERSISTENT
//VAR_GLOBAL
	ProductPar:ST_Parameter;	
	iPersistentDataTese:INT;
	bDataValid:BOOL;//数据有效标志位
END_VAR

// ---- GVLs/GVL_Rectify.TcGVL
VAR_GLOBAL
    arrRecCtrl                : ARRAY[1..MaxRec]  OF  ST_RecCtrl;(*纠偏*)
	AnRecY:ST_RecY;//正极模具
	CaRecY:ST_RecY;//负极模具
END_VAR

VAR_GLOBAL PERSISTENT

END_VAR

VAR_GLOBAL CONSTANT
	  MaxRec			                  	:UINT:=4;		(*纠偏数量*)
END_VAR

// ---- GVLs/GVL_User2.TcGVL
VAR_GLOBAL
		stAnUwindTen		:	ST_Tension;//正极放卷张力
		stAnAuxDriverTen	:	ST_Tension;//正极张力辅助驱动
			
		stCaUwindTen		:	ST_Tension;//负极放卷张力										
		stCaAuxDriverTen	:	ST_Tension;//负极张力辅助驱动
(*
           stAnUwindLTen                                :ST_Tension;//正极张力左放卷
           stAnUwindRTen                             :ST_Tension;//正极张力右放卷
          stAnAuxDriverTen:						ST_Tension;//正极张力辅助驱动			
		   				
           stCaUwindLTen                                :ST_Tension;//负极张力左放卷						
           stCaUwindRTen                             :ST_Tension;//负极张力右放卷						
          stCaAuxDriverTen:						ST_Tension;//负极张力辅助驱动

*)
		
END_VAR

// ---- GVLs/GVL_User3.TcGVL

VAR_GLOBAL


(***方法***)
            stMethod                                 :ST_Method;

            bAllTenReady                              :BOOL;
            bAllGearReady                            :BOOL;
            bAllHomeReady                          :BOOL;


            bAnCamInReady                           :BOOL;
            bCaCamInReady                           :BOOL;

(***条件***)
           bAllTenOk                                   :BOOL;
           bHomeOk                                   :BOOL;        
           bAllGearOK                                :BOOL;
           bAllTempOK                               :BOOL;
           bAllRecOK                                  :BOOL;
           bAllCreatTableOK                        :BOOL;
           bAllCamOK                                 :BOOL;

(**报警**)
         CuterCountAlarm                              :ARRAY[1..8]  OF BOOL;              //切刀计数报警
         arrCYOnAlarm                                :ARRAY[1..MaxCy]  OF BOOL;              //气缸ON报警
         arrCYOFFAlarm                              :ARRAY[1..MaxCy]  OF BOOL;              //气缸OFF报警
         bAnCYHaveAlarm                              :BOOL;                                              //正极气缸有报警
		bCaCYHaveAlarm                              :BOOL;                                              //负极气缸有报警
		
         arrAxisAlarm                                  :ARRAY[1..MaxAxes]  OF BOOL;            //轴报警
         bAnAxisHaveAlarm                              :BOOL;                                             //正极轴有报警
		 bCaAxisHaveAlarm                              :BOOL;                                             //负极轴有报警
		
          bAnTenHaveAlarm                            :BOOL;                                           //正极张力有报警
          bCaTenHaveAlarm                            :BOOL;                                           //负极张力有报警
		  
          
          bAnRecHaveAlarm                            :BOOL;                                          //正极纠偏有报警
          bCaRecHaveAlarm                            :BOOL;                                          //负极纠偏有报警
		         
         bAnCreatTableHaveAlarm                    :BOOL;										//正极创建凸轮有报警
         bCaCreatTableHaveAlarm                    :BOOL;										//负极创建凸轮有报警
		 
         bAnCamHaveAlarm                             :BOOL;										//正极凸轮耦合有报警
         bCaCamHaveAlarm                             :BOOL;										//负极凸轮耦合有报警
		 
         bAnGearHaveAlarm                             :BOOL;										//正极齿轮耦合有报警
         bCaGearHaveAlarm                             :BOOL;										//负极齿轮耦合有报警
		 
         bAnFlowHaveAlarm                             :BOOL;										//正极流程有报警
         bCaFlowHaveAlarm                             :BOOL;										//负极流程有报警

         bAnHaveLightWarn                             :BOOL;										//正极有轻型警告(提示)
         bCaHaveLightWarn                            :BOOL;										//负极有轻型警告(提示)	

		b_lifetime									:BOOL;										//寿命已到	 

		 AnAlarm:ST_AlarmWarn;
		 CaAlarm:ST_AlarmWarn;
		 
		 bAnDoorALM                                :BOOL;                                             //正极门禁先报警
		 bCaDoorALM                                :BOOL;                                             //负极门禁先报警
		 breadALM                                :BOOL;                                             //上电后模切参数读取失败
END_VAR

// ---- GVLs/GCylinder.TcGVL
	
VAR_GLOBAL
	arrCyCtrl			                  :ARRAY[1..MaxCy] OF ST_CyCtrl;	(*气缸控制接口*)
     AA1: INT;
END_VAR

VAR_GLOBAL CONSTANT
	MaxCy			                  	:UINT:=80;		(*气缸数量*)
END_VAR

// ---- GVLs/IO.TcGVL
VAR_GLOBAL
	
//////////////////////////叠片交互////////////////////////////////
AnMQ_MES1	                  AT %Q*    	:ST_BeltData; //叠台1  MES交互
CaMQ_MES1	                  AT %Q*    	:ST_BeltData; //叠台1  MES交互
AnMQ_MES2	                  AT %Q*    	:ST_BeltData; //叠台2  MES交互
CaMQ_MES2	                  AT %Q*    	:ST_BeltData; //叠台2 MES交互
AnMQ_MES3	                  AT %Q*    	:ST_BeltData; //叠台3  MES交互
CaMQ_MES3	                  AT %Q*    	:ST_BeltData; //叠台3  MES交互

//模切、叠台条码交互
	DT_To_MQ_MES AT %I*:ST_DT_To_MQ_MES;
	MQ_To_DT_MES AT %Q*:ST_MQ_To_DT_MES;
//预留数据交互
YL_Q        			AT %Q*:ARRAY[1..50] OF BOOL ; //1、气压不足报警;
YL_I     				AT %I*:ARRAY[1..50] OF BOOL ; //预留输入；
YL_INT1     		AT %Q*:ARRAY[1..50] OF INT  ; //预留输入INT；
YL_INT2     		AT %I*:ARRAY[1..50] OF INT  ; //预留输出INT；
YL_GVL  :ARRAY [1..60] OF BOOL;//内部预留；

//////////////////////////叠片交互////////////////////////////////
D_Pro    AT %I*: DToM_Process;//只读 叠片生产过程信号
D_Sys    AT %I*: DToM_System;//只读 叠片系统信号
M_Pro    AT %Q*: MToD_Process;//只写 模切生产过程信号
M_Sys    AT %Q*: MToD_System;//只写 模切系统信号
MTD_Mes1	 AT %Q*: MTD_Mes1;	//发送模切数据XFP20240315
DTM_Mes1	 AT %I*: DTM_Mes1;	//接收叠台数据XFP20240315

I30101	 AT %I*:BOOL ; //1号叠台:正极模切送料分段皮带1有料感应
I30107	 AT %I*:BOOL ; //1号叠台:负极模切送料分段皮带1有料感应
I40101	 AT %I*:BOOL ; //2号叠台:正极模切送料分段皮带2有料感应
I40107	 AT %I*:BOOL ; //2号叠台:负极模切送料分段皮带2有料感应
I50101	 AT %I*:BOOL ; //3号叠台:正极模切送料分段皮带3有料感应
I50107	 AT %I*:BOOL ; //3号叠台:负极模切送料分段皮带3有料感应

Q30103	 AT %Q*:BOOL;//正极模切分段皮带1除尘毛刷正转
Q30104	 AT %Q*:BOOL;//正极模切分段皮带1除尘毛刷反转
Q30201	 AT %Q*:BOOL;//负极模切分段皮带1除尘毛刷正转
Q30202	 AT %Q*:BOOL;//负极模切分段皮带1除尘毛刷反转

Q40103	 AT %Q*:BOOL;//正极模切分段皮带2除尘毛刷正转
Q40104	 AT %Q*:BOOL;//正极模切分段皮带2除尘毛刷反转
Q40201	 AT %Q*:BOOL;//负极模切分段皮带2除尘毛刷正转
Q40202	 AT %Q*:BOOL;//负极模切分段皮带2除尘毛刷反转

Q50103	 AT %Q*:BOOL;//正极模切分段皮带3除尘毛刷正转
Q50104	 AT %Q*:BOOL;//正极模切分段皮带3除尘毛刷反转
Q50201	 AT %Q*:BOOL;//负极模切分段皮带3除尘毛刷正转
Q50202	 AT %Q*:BOOL;//负极模切分段皮带3除尘毛刷反转


/////////////////////////正极模切/////////////////////
I101      AT %I*:ARRAY[1..16] OF BOOL ;  	//输入模块
I102		AT %I*:ARRAY[1..16] OF BOOL ;  	//输入模块
I103		AT %I*:ARRAY[1..16] OF BOOL ;  	//输入模块
I104		AT %I*:ARRAY[1..16] OF BOOL ;  	//输入模块
I105		AT %I*:ARRAY[1..16] OF BOOL ;  	//输入模块
I106		AT %I*:ARRAY[1..16] OF BOOL ;  	//输入模块
I107		AT %I*:ARRAY[1..16] OF BOOL ;  	//输入模块
I108		AT %I*:ARRAY[1..16] OF BOOL ;  	//输入模块
I109		AT %I*:ARRAY[1..16] OF BOOL ;  	//输入模块

Q101		AT %Q*:ARRAY[1..16] OF BOOL ;  	//输出模块
Q102		AT %Q*:ARRAY[1..16] OF BOOL ;  	//输出模块
Q103		AT %Q*:ARRAY[1..16] OF BOOL ;  	//输出模块
Q104		AT %Q*:ARRAY[1..16] OF BOOL ;  	//输出模块
Q105		AT %Q*:ARRAY[1..16] OF BOOL ;  	//输出模块
Q106		AT %Q*:ARRAY[1..16] OF BOOL ;  	//输出模块
Q107		AT %Q*:ARRAY[1..16] OF BOOL ;  	//输出模块
Q108		AT %Q*:ARRAY[1..16] OF BOOL ;  	//输出模块
Q109		AT %Q*:ARRAY[1..16] OF BOOL ;  	//输出模块

AI101	AT %I*:ARRAY[0..3]    OF INT;  //模拟量输入
AI102	AT %I*:ARRAY[0..3]    OF INT;  //模拟量输入

AO101  AT %Q*:ARRAY[0..3]   OF INT;  //模拟量输出

/////////////////////////负极模切/////////////////////
I201      AT %I*:ARRAY[1..16] OF BOOL ;  	//输入模块
I202		AT %I*:ARRAY[1..16] OF BOOL ;  	//输入模块
I203		AT %I*:ARRAY[1..16] OF BOOL ;  	//输入模块
I204		AT %I*:ARRAY[1..16] OF BOOL ;  	//输入模块
I205		AT %I*:ARRAY[1..16] OF BOOL ;  	//输入模块
I206		AT %I*:ARRAY[1..16] OF BOOL ;  	//输入模块
I207		AT %I*:ARRAY[1..16] OF BOOL ;  	//输入模块
I208		AT %I*:ARRAY[1..16] OF BOOL ;  	//输入模块
I209		AT %I*:ARRAY[1..16] OF BOOL ;  	//输入模块

Q201		AT %Q*:ARRAY[1..16] OF BOOL ;  	//输出模块
Q202		AT %Q*:ARRAY[1..16] OF BOOL ;  	//输出模块
Q203		AT %Q*:ARRAY[1..16] OF BOOL ;  	//输出模块
Q204		AT %Q*:ARRAY[1..16] OF BOOL ;  	//输出模块
Q205		AT %Q*:ARRAY[1..16] OF BOOL ;  	//输出模块
Q206		AT %Q*:ARRAY[1..16] OF BOOL ;  	//输出模块
Q207		AT %Q*:ARRAY[1..16] OF BOOL ;  	//输出模块
Q208		AT %Q*:ARRAY[1..16] OF BOOL ;  	//输出模块
Q209		AT %Q*:ARRAY[1..16] OF BOOL ;  	//输出模块

AI201	AT %I*:ARRAY[0..3]    OF INT;  //模拟量输入
AI202	AT %I*:ARRAY[0..3]    OF INT;  //模拟量输入

AO201  AT %Q*:ARRAY[0..3]   OF INT;  //模拟量输出
	
/////////////////////////////////////////////////////////////////////////////////////////////////////////////////////////////
   AnBtn                  :ST_MoQieButton;//正极
   CaBtn                  :ST_MoQieButton;//负极
   AnSenser             :ST_MoQieSenser;//正极
   CaSenser             :ST_MoQieSenser;//负极

END_VAR

VAR_GLOBAL CONSTANT
	MaxAINo				:INT:=24;		(*ai通道数量*)
END_VAR

// ---- GVLs/GMotion.TcGVL
	
VAR_GLOBAL
	arrAxis			                      :ARRAY[1..MaxAxes] OF  axis_ref;		(*PTP轴*)
	arrAxisCtrl			                  :ARRAY[1..MaxAxes] OF ST_AxisCtrl;	(*轴的PTP控制接口*)
    AnSetpMotor               : ST_SetpMotor;//正极NG收料排杆电机
    CaSetpMotor              : ST_SetpMotor;//负极NG收料排杆电机
	arrDustMotor			                      :ARRAY[1..MaxDust] OF  ST_DustMotor;		(*毛刷电机*)
    AxisCtrlTest                           AT%Q*:  ST_AxisCtrl;

	 DrivesOP 		                       AT %I*		:ARRAY[1..NumOfDrives	]OF UINT ;		                                 (*实际驱动器作为EtherCAT伺服的个数  ETHERCAT状态*)

	iActDriveMode	                   AT%I*	    	:ARRAY[1..2]OF SINT;			                                 (*驱动器返回的控制模式*)
	iActDriveTorque	                   AT%I*	    	:ARRAY[1..2]OF INT;			                                 (*驱动器返回的l力矩*)

    iSetDriveMode 	                  AT %Q*    	:ARRAY [1..2] OF SINT := [10,10] ;         // (*驱动器的模式输出，8为位置模式*)

	iMaxProfileVelo                   AT%Q* 	   :ARRAY[1..2]OF UDINT:=[139810133,139810133];    //   (*单位为0.1rpm  500*2(23)   *)\
	iPostiveTorqueLimits            AT%Q* 	  :ARRAY[1..2]OF UINT:=[2000,2000];
    iNegtiveTorqueLimits           AT%Q*     :ARRAY[1..2]OF UINT:=[2000,2000];
	
	iActTorque_M				AT%I*	    	:ARRAY[1..MaxAxes]OF INT;	//模切轴反馈力矩值
	HMI_TorAlarm_M				:ARRAY[1..MaxAxes]OF BOOL ;	//模切轴反馈力矩过大报警(防止撞机)
	HMI_MS_Speed				:ARRAY[1..20]OF REAL ;	//毛刷转速
END_VAR

VAR_GLOBAL CONSTANT
	MaxAxes				:UINT:=60;		(*NC轴数，不同于实轴数*)
    NumOfDrives			:UINT:=48;		(*实轴数*)
	iEcatOp			     	:UINT:=8;
	CSP					    :USINT:=8;
	CSV					    :USINT:=9;
	CST					    :USINT:=10;
	MaxDust               	:UINT:=20;
END_VAR

VAR_GLOBAL PERSISTENT
//VAR_GLOBAL
	arrAxisPar		   	:ARRAY[1..MaxAxes] OF ST_Axis_Par;	(*轴的PTP控制接口*)
    iTargetTorque	                  AT%Q*    	:ARRAY[1..2]OF INT:= [10,10];			                     (*单位为0.1%*) //最大为100
	HMI_TorErrLimt_M				:ARRAY[1..MaxAxes]OF INT:=[MaxAxes(2000)]  ;	//模切轴反馈力矩报警上限值设定,初始设定值2000
END_VAR















	//aAxis_NcParam			:ARRAY[1..MaxAxes] OF ST_AxisParameterSet;	(*system manager中的NC参数读取*)
	//aReadNcParam			:ARRAY[1..MaxAxes] OF MC_ReadParameterSet; //FB
	//aWriteNcParam	        :ARRAY[1..MaxAxes] OF MC_WriteParameter;  //system manager中的NC参数写入
    //  mc_AxisParameter2       :E_AxisWritePar;




(************************************************************************************)
	(*欧姆龙驱动器力矩模式
	输出：
		6071 目标扭矩  INT16    0.1%  -5000~5000   （建议设置为PDO
		6072 最大扭矩 UINT16    0.1%  0~5000		（建议在驱动器中设置好
		3031 -01  力矩模式下的速度限制 单位rpm ，0-20000  INT32   出厂20000
	输入：当前力矩 6072
	*)
	(*
(*0821增加张力伺服参数*)
	iTartgetTorque	AT%Q*:ARRAY[2..2]OF INT:=[-80,80];		(*单位为0.1%*)
	iMaxVelo		AT%Q*:ARRAY[2..2]OF UDINT:=NumOfDancers[8000];	(*单位为0.1rpm*)
	iActualTorque	AT%I* :ARRAY[2..2]OF  INT;							(*单位为0.1%*)
	iSetDriveMode 	AT %Q*		:ARRAY [1..NumOfDrives] OF SINT := NumOfDrives[CSP];	(*驱动器的模式输出，8为位置模式*)
*)

// ---- GVLs/N.TcGVL
VAR_GLOBAL  PERSISTENT//断电保持
(*(**轴**)
	AnAxisNo:      ST_AxisName;  //正极
	CaAxisNo:      ST_AxisName;//负极
	
    AnVirAxisNo:      ST_VirAxisName;//正极
	CaVirAxisNo:      ST_VirAxisName;//负极
	VirTimeWind:INT;//模切虚拟摆杆放卷轴 
(**气缸**)
	AnCYNo:        ST_CylinderName;//正极
	CaCYNo:        ST_CylinderName;//负极

(**电磁阀**)
	AnEVNo:        ST_ElectValveName;//正极
	CaEVNo:        ST_ElectValveName;//负极

(***纠偏**)
    AnRecNo:         ST_RecName;//正极
	CaRecNo:         ST_RecName;//负极

(***凸轮表号**)
	 AnTableNo:  ST_TableNo;// 正极
	 CaTableNo:  ST_TableNo;// 负极
	 
(***除尘电机号**)
	 AnMotorNo:  ST_MotorName;// 正极
	 CaMotorNo:  ST_MotorName;// 负极
	 *)
	NameNo:ST_Name;
END_VAR

// ---- GVLs/System.TcGVL

VAR_GLOBAL	
	stHmiSysCmd			    	    :ST_SysCmd;
	MachimeVersion				:STRING:='V2024.5.28';(*当前系统版本号*)
	MachimeTpye					:STRING:='YKRFH';
	SysInfo						       :SystemInfoCtrl;
	fPlcCycleTime_ms			    :LREAL;
	pulse						            :PulseCtrl;	
	stTime: TIMESTRUCT;
	versionwrite  : BOOL;//版本号写入
END_VAR

// ---- GVLs/User01.TcGVL

VAR_GLOBAL
	 stSysState :ST_SystemPublic;//系统状态机(整机公用)
	 AnSys:ST_SystemPart;//系统状态机(正极)
	 CaSys:ST_SystemPart;//系统状态机(负极)
	 P2Interaction:ST_P2InteractPub;//叠片公共交互
	 AnInter:ST_P2InteractPart;//正极交互
	 CaInter:ST_P2InteractPart;//负极交互
	 AnCCDCom:ST_CCDCom;
	 CaCCDCom:st_CCDCom;
	 AnCCDIO:ST_CCDIO;
	 CaCCDIO:st_CCDIO;
      arrda1:                         UINTARR2;
      fbPulseCtrl                  :ARRAY[1..10]   OF      PulseGeneratorCtrl;
	  bytePower: BYTE:=16#01;
	  
	PLC_wYear:UINT;//PLC时间年
	PLC_wMonth:UINT;//PLC时间月
	PLC_wDay:UINT;//PLC时间日
	PLC_wHour:UINT;//PLC时间时
	PLC_wMinute:UINT;//PLC时间分
	PLC_wSecond:UINT;//PLC时间秒
	PLC_wMilliseconds:WORD;//PLC时间毫秒
	AnSysNgMark:ST_NGMark;
	CaSysNgMark:ST_NGMark;
	fbAnProductLocal: ProductLocal;
	fbCaProductLocal: ProductLocal;
	
	MQQuery:BOOL;//时间查询
	MQdate:INT;//查询日期
	
	MQ_Mes1	:DTM_Mes1;	//XFP20240315
END_VAR


VAR_GLOBAL PERSISTENT
	An_Production	:LocalProduction; //正极产能；
	Ca_Production	:LocalProduction;//负极产能；
	//aAnDay_date: Day_date; //正极产能；
	//aCaDay_date: Day_date; //负极产能；
	Antimedata:FB_DataTime;//运行时间
	Catimedata:FB_DataTime;//运行时间
	cCn_An:REAL;
	cCn_Ca:REAL;
	PoleData:ST_Data;
	AnMQ_FingerprintKey:ST_FingerprintKey; //指纹解锁	 
	CaMQ_FingerprintKey:ST_FingerprintKey; //指纹解锁		 
 	YL_GVL2: ARRAY [1..60] OF DINT ;//内部预留；//  1、正极R角已经切的次数;  2、正极R角设置清废报警次数；3、负极R角已经切的次数;  4、负极R角设置清废报警次数；
	CS:ARRAY[0..2] OF INT;//切刀报警角度调整；
(*产能统计*)	
	HMI_AnTodayNGClass_AM		:ARRAY[1..30 ] 	OF REAL;(*当天白班各类NG数量ARRAY[1..30 ]-----正极*)
	HMI_AnTodayNGClass_PM		:ARRAY[1..30 ] 	OF REAL;(*当天夜班各类NG数量ARRAY[1..30 ]-----正极*)
	HMI_AnTodayNG_AM:REAL;(*当天白班生产NG总数-----正极*)
	HMI_AnTodayNG_PM:REAL;(*当天夜班生产NG总数-----正极*)
	
	HMI_CaTodayNGClass_AM		:ARRAY[1..30 ] 	OF REAL;(*当天白班各类NG数量ARRAY[1..30 ]-----负极*)
	HMI_CaTodayNGClass_PM		:ARRAY[1..30 ] 	OF REAL;(*当天夜班各类NG数量ARRAY[1..30 ]-----负极*)
	HMI_CaTodayNG_AM:REAL;(*当天白班生产NG总数-----负极*)
	HMI_CaTodayNG_PM:REAL;(*当天夜班生产NG总数-----负极*)
END_VAR


VAR_GLOBAL CONSTANT
     	DD2: INT := 1;
		//PI:REAL:=3.1415926;
END_VAR


































	(* 
  
   	 scRecipe :            CS_Recipe;
	 iRecipe:               IRecipe;
	 arriVirSingle:    ARRAY  [1..30] OF INT:=[30(1)] ;  //虚拟仿真信号
	 arriVirSingle2:  ARRAY [1..30] OF INT:=[30(1)] ;  //虚拟仿真信号
	 arriVirSingle3:  ARRAY [1..30] OF INT:=[30(1)] ;  //虚拟仿真信号


	arrAxisError :                ARRAY[1..MaxAxes] OF BOOL;//轴报警
	arrActuatorsError :        ARRAY[1..20] OF BOOL;//气缸
	arrFunctionError :         ARRAY[1..20] OF BOOL;//功能


	 cmd: CMD;
	 ShortDataShow:ShortDataShow; 
	 csShortTest :CS_ShortTest;
	 csCodeTcp: CS_CodeTcp;
	 IShort:IShortTest;
	 iCode:ICode;
	csCcdTcp:CS_CcdTcp_V2;
	iCCD:ICCD;
	ccdData:STCcdData;
	*)

// ---- POUs/POUs/MAIN.TcPOU
PROGRAM MAIN
VAR
	BUSY: BOOL;
	ERR: BOOL;
	ERRID: UDINT;
	CSData:    CS_Data;
	

	THNN: INT;
	MA100: BOOL;
	A1: BOOL;
	D1: BOOL;
	A2: BOOL;
	A3: BOOL;
	
	//iShort:        IShortTest;
	D2: INT;
	//stTime: TIMESTRUCT;
	strTime: STRING;
	BY1:  BYTE;
	AA1: BOOL;
	btest: BOOL;
	iPower: INT;
	iPowerSetp: INT;
	boPower2: BOOL;
	k: INT:=1;
	PowerOnDone: BOOL;
	
   tRead			:TON;
END_VAR

VAR
	bFirstCycle										        	:BOOL;	(*初始化用的*)
(*保存掉电保持参数*)
	FB_WritePersistentData1								: FB_WritePersistentData;
	tCycleTimer											: TON;
	bWrite												: BOOL;    (*定时自动保存*)
(*系统重启*)
	tNtDelayReset										:TON;
	bReboot											: BOOL;	(*重启系统的变量*)
	NT_Reboot1											: NT_Reboot;
(*系统关机*)
	NT_Shutdown1										: NT_Shutdown;
	tNtDelayShutdown									: TON;
	bShutdown											: BOOL;
(*远程桌面接管*)
	OpenRemoteDesktop									: NT_StartProcess;
	timerHMI											:TON;
(*系统时间获取*)
	NT_GetTime1											: NT_GetTime;
(*心跳信号*)
	bHeartBeat											:BOOL;
	tHeartBeatTime										:TIME:=t#0.5s;
	TonHeartBeat										:TON;

	TaskInfo											:	TaskInfoCtrl;
	loadParaStep: UINT;
	i: UINT;	

    tonPowerOn  :Tc2_Standard.TON;
    tonPower       :Tc2_Standard.TON;


     STR1: STRING:='20200412160000';
	 STR2: STRING:='12345678ABCDE';
	 STR3: STRING:='SSDDFF1234  JJJJ';
	 size:UDINT;
	 
	rt:ARRAY[1..10]OF R_TRIG;//上升沿触发
	ft:ARRAY[1..10]OF F_TRIG;//下降沿触发
	testii2: INT;
	bReadDataFirstCyle: BOOL;
	bReadDataCyle2: BOOL;
	bSaveTest: BOOL;
	rtSaveData: R_TRIG;
	fbDataXML       : FB_DataXML;//XML参数保存功能块
	rt10:Tc2_Standard.R_TRIG;
	testii:INT:=0;
	 
END_VAR

(*===========================================版本号=================================================*)
//MachimeVersion:='V3.0-24/3/2';(*HMI显示当前程序版本号*)
IF versionwrite THEN
   MachimeVersion:=CONCAT(CONCAT(CONCAT(CONCAT('V',CONCAT( WORD_TO_STRING(stTime.wYear),'.')),WORD_TO_STRING(stTime.wMonth)),'.'),WORD_TO_STRING(stTime.wDay));
END_IF
(*
版本： 

((*
1、线扫OK与NG信号IO触发;（02.20）
2、叠台NG梯度踢废空叠隔膜程序；（02.20）
3、叠台NG梯度踢废下料方式程序；（02.20）
4、隔膜剩余长度计算程序;（02.21）
5、无极片编号传送带尾部排废程序；（02.23）
6、对齐度NG计数程序  （02.27）
7、接带后找极耳程序；（02.28）
8、模切风刀吹气程序；（3.2）
9、程序版本号程序；（3.2）
10、叠台搬运极耳真空检测程序；（3.3）
11、冷压扫二维码程序；（3.3）
12、隔膜剩余长度计算（通过卷径大小）程序;（03.3）
13、隔膜卷径报警值限定（93），卷径报警实时判断改为叠完一个电芯判断一次;（03.6）
14、叠台搬运和压刀凸轮曲线修改，压刀升降和压刀开合行程限定；（03.12）
15、模切线扫结果判定逻辑优化，线扫触发和结果计数；（03.12）
16、新增模切放卷尾料4连标程序；（03.13）
17、模切黄标和接带踢废程序优化；（03.13）
18、短卷针回零增加安全条件(短卷针旋转轴原点传感器需亮)；（03.13）
19、模切放卷激光器继电器控制启用；（3.17）
20、触摸屏门禁屏蔽取消；（3.17）
21、增加启动CCD自检弹窗，需要确认后才能启动；（3.26）
22、叠台气涨轴开关有信号，隔膜踢废；（3.26）
23、触摸屏三级权限；（3.26）
24、上位机优率表；（3.31）
25、黄标跳切计数；（3.26）
26、黄标计数；（4.1）
27、叠台增加调试模式；（4.2）
28、热切丝寿命计数；（4.2）
29、模切尾料四连标检测；（4.2）
30、对齐度单片踢废；（4.5）
31、隔膜尾料角度计算；（4.5）
32、断带后R角不冲切；（4.7）
33、黄标与接带感应后日志；（4.7）
34、极片间距报警；（4.17）
35、凸轮位置角度固定；（4.17）
36、空叠首尾层隔膜降速降张力；（4.17）
37、正极真空改成常开；（4.17）
38、纠偏台重复精度测试；（4.17）
39、二维码贴胶完成自动备胶默停、重胶；（4.20）
40、对齐度踢废后第一片纠偏平台不纠偏；（4.20）
41、叠台一键初始化；（4.20）
42、模切尺寸、倒装、分段皮带比例系数改成一致；（4.20）
43、尾卷纠偏到限位，凸轮耦合报警；（4.20）
44、叠最后一层隔膜负极叠台升降放片位置下降少一点；（4.20）
45、模切R角横深纵深闭环纠偏；（4.20）
46、CCD标定与重复精度测试电机到位后延时拍照；（4.20）
47、短卷针夹泄气真空；（4.21）
48、对齐度闭环纠偏；（4.21）
49、模切触发高速停止；（4.22）
50、叠片取分段皮带取料中信号提前复位；（4.22）
51、贴胶头进退增加软限位；（4.23）
52、叠台0步增加判断，正负极不能执行同时往叠台方向运动流程；（4.23）
53、热压一键初始化；（4.23）
*)
   
*)
(*====================================================================================================*)



TwinCAT_Nt();

Main.XML();






tonPowerOn(IN:=PowerOnDone , PT:=T#5S , Q=> , ET=> );  //上电延时3S
IF PowerOnDone THEN
 IOLink();
END_IF

IF tonPowerOn.Q AND fbDataXML.bReadParDone THEN
 MainState();
 FingerprintKey();  
;
;
ELSE
	;
   Power();//接触器上电
END_IF




AA1;

//字体设置成中文字体  解决了注释乱码的问题






// scRecipe(iRecipe2:=iRecipe );
 







 //正极NG类型计数
 fbAnProductLocal(
	NGFlag1:=AnSysNgMark.NGMark[1] , 
	NGFlag2:=AnSysNgMark.NGMark[2], 
	NGFlag3:=AnSysNgMark.NGMark[3], 
	NGFlag4:=AnSysNgMark.NGMark[4] , 
	NGFlag5:=AnSysNgMark.NGMark[5] , 
	NGFlag6:=AnSysNgMark.NGMark[6] , 
	NGFlag7:=AnSysNgMark.NGMark[7] , 
	NGFlag8:=AnSysNgMark.NGMark[8] , 
	NGFlag9:=AnSysNgMark.NGMark[9] , 
	NGFlag10:=AnSysNgMark.NGMark[10] , 
	NGFlag11:=AnSysNgMark.NGMark[11] , 
	NGFlag12:=AnSysNgMark.NGMark[12] , 
	NGFlag13:=AnSysNgMark.NGMark[13], 
	NGFlag14:=AnSysNgMark.NGMark[14] , 
	NGFlag15:=AnSysNgMark.NGMark[15] , 
	NGFlag16:=AnSysNgMark.NGMark[16] , 
	NGFlag17:=AnSysNgMark.NGMark[17] , 
	NGFlag18:=AnSysNgMark.NGMark[18] , 
	NGFlag19:=AnSysNgMark.NGMark[19] , 
	NGFlag20:=AnSysNgMark.NGMark[20] , 
	NGFlag21:=AnSysNgMark.NGMark[21] , 
	NGFlag22:=AnSysNgMark.NGMark[22] , 
	NGFlag23:=AnSysNgMark.NGMark[23] , 
	NGFlag24:=AnSysNgMark.NGMark[24] , 
	NGFlag25:=AnSysNgMark.NGMark[25] , 
	NGFlag26:=AnSysNgMark.NGMark[26] , 
	NGFlag27:=AnSysNgMark.NGMark[27] , 
	NGFlag28:=AnSysNgMark.NGMark[28] , 
	NGFlag29:=AnSysNgMark.NGMark[29] , 
	NGFlag30:=AnSysNgMark.NGMark[30] , 
	TodayNGClass_AM=>HMI_AnTodayNGClass_AM, (*当天白班各类NG数量ARRAY[1..30 ]*)
	TodayNGClass_PM=>HMI_AnTodayNGClass_PM , (*当天夜班各类NG数量ARRAY[1..30 ]*)
	TodayNG_AM=>HMI_AnTodayNG_AM , (*当天白班生产NG总数*)
	TodayNG_PM=>HMI_AnTodayNG_PM );(*当天夜班生产NG总数*)

 
 
 
 //负极NG类型计数
fbCaProductLocal(
	NGFlag1:=CaSysNgMark.NGMark[1] , 
	NGFlag2:=CaSysNgMark.NGMark[2], 
	NGFlag3:=CaSysNgMark.NGMark[3], 
	NGFlag4:=CaSysNgMark.NGMark[4] , 
	NGFlag5:=CaSysNgMark.NGMark[5] , 
	NGFlag6:=CaSysNgMark.NGMark[6] , 
	NGFlag7:=CaSysNgMark.NGMark[7] , 
	NGFlag8:=CaSysNgMark.NGMark[8] , 
	NGFlag9:=CaSysNgMark.NGMark[9] , 
	NGFlag10:=CaSysNgMark.NGMark[10] , 
	NGFlag11:=CaSysNgMark.NGMark[11] , 
	NGFlag12:=CaSysNgMark.NGMark[12] , 
	NGFlag13:=CaSysNgMark.NGMark[13], 
	NGFlag14:=CaSysNgMark.NGMark[14] , 
	NGFlag15:=CaSysNgMark.NGMark[15] , 
	NGFlag16:=CaSysNgMark.NGMark[16] , 
	NGFlag17:=CaSysNgMark.NGMark[17] , 
	NGFlag18:=CaSysNgMark.NGMark[18] , 
	NGFlag19:=CaSysNgMark.NGMark[19] , 
	NGFlag20:=CaSysNgMark.NGMark[20] , 
	NGFlag21:=CaSysNgMark.NGMark[21] , 
	NGFlag22:=CaSysNgMark.NGMark[22] , 
	NGFlag23:=CaSysNgMark.NGMark[23] , 
	NGFlag24:=CaSysNgMark.NGMark[24] , 
	NGFlag25:=CaSysNgMark.NGMark[25] , 
	NGFlag26:=CaSysNgMark.NGMark[26] , 
	NGFlag27:=CaSysNgMark.NGMark[27] , 
	NGFlag28:=CaSysNgMark.NGMark[28] , 
	NGFlag29:=CaSysNgMark.NGMark[29] , 
	NGFlag30:=CaSysNgMark.NGMark[30] , 
	TodayNGClass_AM=> HMI_CaTodayNGClass_AM, (*当天白班各类NG数量ARRAY[1..30 ]*)
	TodayNGClass_PM=>HMI_CaTodayNGClass_PM , (*当天夜班各类NG数量ARRAY[1..30 ]*)
	TodayNG_AM=>HMI_CaTodayNG_AM , (*当天白班生产NG总数*)
	TodayNG_PM=>HMI_CaTodayNG_PM );(*当天夜班生产NG总数*)

ACTION Power:
(***系统延时启动***)

tonPower(IN:= , PT:=T#1.5S , Q=> , ET=> );

CASE iPowerSetp OF
0:
    tonPower.IN:=TRUE;
    iPowerSetp:=10;
10:
   IF   tonPower.Q  THEN
      bytePower:=SHL(bytePower,1);
     
      tonPower(IN:=FALSE );
      k:=k+1;
     iPowerSetp:=20;
  END_IF
20:
    bytePower.0:=1;
    tonPower.IN:=TRUE;
    iPowerSetp:=30;
30:
   IF  k>=8 THEN
        iPowerSetp:=40;
       // bytePower:=16#00;
        //PowerOnDone:=TRUE;
   ELSE
      iPowerSetp:=10;
   END_IF
  40:
  	(********************** Name赋值   ***************************************)
	//////轴号//////					
NameNo.	AnAxisNo.	UnWind_L	:=	1	;//模切左放卷	
NameNo.	AnAxisNo.	UnWind_R	:=	2	;//模切右放卷	
NameNo.	AnAxisNo.	PoleTension	:=	3	;//模切前摆杆张力	
NameNo.	AnAxisNo.	DriverAux	:=	4	;//模切辅助驱动	
NameNo.	AnAxisNo.	BuffeLine	:=	5	;//模切极片缓存	
NameNo.	AnAxisNo.	Mould	:=	6	;//倒角模具	
NameNo.	AnAxisNo.	MouldRectify_X	:=	7	;//模具纠偏X轴(肩宽补偿)	
NameNo.	AnAxisNo.	MouldRectify_Y	:=	8	;//模具纠偏Y轴(切刀深度)	
NameNo.	AnAxisNo.	DriverDDR	:=	9	;//模切主驱动	
NameNo.	AnAxisNo.	Cuter	:=	10	;//裁切切刀	
NameNo.	AnAxisNo.	CuterDegRectify	:=	11	;//裁切角度纠偏	
NameNo.	AnAxisNo.	CuterBelt	:=	12	;//裁切输送皮带	
NameNo.	AnAxisNo.	CuterBeltChange	:=	13	;//裁切输送带换型	
NameNo.	AnAxisNo.	CCDPressPush	:=	14	;//尺寸CCD压片升降	
NameNo.	AnAxisNo.	NGPushReverseBelt	:=	15	;//踢废倒装皮带	
NameNo.	AnAxisNo.	NGPush1	:=	16	;//踢连续废料	
NameNo.	AnAxisNo.	NGPush2	:=	17	;//踢单张废料	
NameNo.	AnAxisNo.	DedustBelt	:=	18	;//上表面除尘皮带	
NameNo.	AnAxisNo.	DedustReverseBelt	:=	19	;//下表面除尘倒装皮带	
NameNo.	AnAxisNo.	SubBelt1	:=	20	;//送料分段皮带1	
NameNo.	AnAxisNo.	SubBelt2	:=	21	;//送料分段皮带2	
NameNo.	AnAxisNo.	SubBelt3	:=	22	;//送料分段皮带3	
NameNo.	AnAxisNo.	Ready1	:=	23	;//备用1	
NameNo.	AnAxisNo.	Ready2	:=	24	;//备用2	
						
NameNo.	CaAxisNo.	UnWind_L	:=	25	;//模切左放卷	
NameNo.	CaAxisNo.	UnWind_R	:=	26	;//模切右放卷	
NameNo.	CaAxisNo.	PoleTension	:=	27	;//模切前摆杆张力	
NameNo.	CaAxisNo.	DriverAux	:=	28	;//模切辅助驱动	
NameNo.	CaAxisNo.	BuffeLine	:=	29	;//模切极片缓存	
NameNo.	CaAxisNo.	Mould	:=	30	;//倒角模具	
NameNo.	CaAxisNo.	MouldRectify_X	:=	31	;//模具纠偏X轴(肩宽补偿)	
NameNo.	CaAxisNo.	MouldRectify_Y	:=	32	;//模具纠偏Y轴(切刀深度)	
NameNo.	CaAxisNo.	DriverDDR	:=	33	;//模切主驱动	
NameNo.	CaAxisNo.	Cuter	:=	34	;//裁切切刀	
NameNo.	CaAxisNo.	CuterDegRectify	:=	35	;//裁切角度纠偏	
NameNo.	CaAxisNo.	CuterBelt	:=	36	;//裁切输送皮带	
NameNo.	CaAxisNo.	CuterBeltChange	:=	37	;//裁切输送带换型	
NameNo.	CaAxisNo.	CCDPressPush	:=	38	;//尺寸CCD压片升降	
NameNo.	CaAxisNo.	NGPushReverseBelt	:=	39	;//踢废倒装皮带	
NameNo.	CaAxisNo.	NGPush1	:=	40	;//踢连续废料	
NameNo.	CaAxisNo.	NGPush2	:=	41	;//踢单张废料	
NameNo.	CaAxisNo.	DedustBelt	:=	42	;//上表面除尘皮带	
NameNo.	CaAxisNo.	DedustReverseBelt	:=	43	;//下表面除尘倒装皮带	
NameNo.	CaAxisNo.	SubBelt1	:=	44	;//送料分段皮带1	
NameNo.	CaAxisNo.	SubBelt2	:=	45	;//送料分段皮带2	
NameNo.	CaAxisNo.	SubBelt3	:=	46	;//送料分段皮带3	
NameNo.	CaAxisNo.	Ready1	:=	47	;//备用1	
NameNo.	CaAxisNo.	Ready2	:=	48	;//备用2	
						
NameNo.	VirTimeWind:=50;//虚拟放卷TIme轴					
						
NameNo.	AnVirAxisNo.VirMain:=51;//模切虚拟主轴					
NameNo.	AnVirAxisNo.VirDriver:=52;//模切虚拟驱动辊					
NameNo.	AnVirAxisNo.VirBelt:=53;//模切虚拟皮带轴					
						
NameNo.	CaVirAxisNo.VirMain:=56;//模切虚拟主轴					
NameNo.	CaVirAxisNo.VirDriver:=57;//模切虚拟驱动辊					
NameNo.	CaVirAxisNo.VirBelt:=58;//模切虚拟皮带轴					
						
	//////气缸和阀号//////					
NameNo.	AnCYNo.	Inflation_L	:=	1	;(*左放卷气胀轴气缸*)	
NameNo.	AnCYNo.	Inflation_R	:=	2	;(*右放卷气胀轴气缸*)	
NameNo.	AnCYNo.	BoardPressL	:=	3	;(*左接带压板气缸*)	
NameNo.	AnCYNo.	BoardPressR	:=	4	;(*右接带压板气缸*)	
NameNo.	AnCYNo.	DriverPressAux	:=	5	;(*辅助驱动压辊气缸*)	
NameNo.	AnCYNo.	CoderRollPress	:=	6	;(*编码器辊压辊气缸*)	
NameNo.	AnCYNo.	DriverPressDDR	:=	7	;(*主驱动压辊气缸*)	
NameNo.	AnCYNo.	NGRevBeltUpDown	:=	8	;(*踢废倒装皮带升降气缸*)	
NameNo.	AnCYNo.	NGRevBeltTension	:=	9	;(*踢废倒装皮带张紧气缸*)	
NameNo.	AnCYNo.	PoleBrushDustPush_U	:=	11	;(*极片上表面毛刷除尘升降缸*)	
NameNo.	AnCYNo.	PoleWindDustPush_U	:=	12	;(*极片上表面风刀除尘升降缸*)	
NameNo.	AnCYNo.	PoleBrushDustPush_D	:=	13	;(*极片下表面毛刷除尘升降缸*)	
NameNo.	AnCYNo.	PoleWindDustPush_D	:=	14	;(*极片下表面风刀除尘升降缸*)	
NameNo.	AnCYNo.	DustRevBeltUpDown	:=	15	;(*极片下表面除尘倒装皮带升降气缸*)	
NameNo.	AnCYNo.	NGBoxLock1	:=	16	;(*NG料盒归正气缸1*)	
NameNo.	AnCYNo.	NGBoxLock2	:=	17	;(*NG料盒归正气缸2*)	
NameNo.	AnCYNo.	WasteBoxPush	:=	18	;(*连续废料收集箱推料气缸*)	
						
NameNo.	CaCYNo.	Inflation_L	:=	21	;(*左放卷气胀轴气缸*)	
NameNo.	CaCYNo.	Inflation_R	:=	22	;(*右放卷气胀轴气缸*)	
NameNo.	CaCYNo.	BoardPressL	:=	23	;(*左接带压板气缸*)	
NameNo.	CaCYNo.	BoardPressR	:=	24	;(*右接带压板气缸*)	
NameNo.	CaCYNo.	DriverPressAux	:=	25	;(*辅助驱动压辊气缸*)	
NameNo.	CaCYNo.	CoderRollPress	:=	26	;(*编码器辊压辊气缸*)	
NameNo.	CaCYNo.	DriverPressDDR	:=	27	;(*主驱动压辊气缸*)	
NameNo.	CaCYNo.	NGRevBeltUpDown	:=	28	;(*踢废倒装皮带升降气缸*)	
NameNo.	CaCYNo.	NGRevBeltTension	:=	29	;(*踢废倒装皮带张紧气缸*)	
NameNo.	CaCYNo.	PoleBrushDustPush_U	:=	31	;(*极片上表面毛刷除尘升降缸*)	
NameNo.	CaCYNo.	PoleWindDustPush_U	:=	32	;(*极片上表面风刀除尘升降缸*)	
NameNo.	CaCYNo.	PoleBrushDustPush_D	:=	33	;(*极片下表面毛刷除尘升降缸*)	
NameNo.	CaCYNo.	PoleWindDustPush_D	:=	34	;(*极片下表面风刀除尘升降缸*)	
NameNo.	CaCYNo.	DustRevBeltUpDown	:=	35	;(*极片下表面除尘倒装皮带升降气缸*)	
NameNo.	CaCYNo.	NGBoxLock1	:=	36	;(*NG料盒归正气缸1*)	
NameNo.	CaCYNo.	NGBoxLock2	:=	37	;(*NG料盒归正气缸2*)	
NameNo.	CaCYNo.	WasteBoxPush	:=	38	;(*连续废料收集箱推料气缸*)	
						
NameNo.	AnEVNo.	ConnectDustVacuo	:=	41	;	//
NameNo.	AnEVNo.	LineSceneDustBlow	:=	42	;	//
NameNo.	AnEVNo.	LineSceneDustVacuo	:=	43	;	//
NameNo.	AnEVNo.	AreaArrayDustBlow	:=	44	;	//
NameNo.	AnEVNo.	MouldUpBlow	:=	45	;	//
NameNo.	AnEVNo.	MouldDownVacuo	:=	46	;	//
NameNo.	AnEVNo.	MouldDownAir	:=	47	;	//
NameNo.	AnEVNo.	NGPushInsideAir	:=	48	;	//
NameNo.	AnEVNo.	NGPushInsideVacuo	:=	49	;	//
NameNo.	AnEVNo.	BrushDustVacuo_U	:=	50	;	//
NameNo.	AnEVNo.	WindDustBlow_U	:=	51	;	//
NameNo.	AnEVNo.	WindDustVacuo_U	:=	52	;	//
NameNo.	AnEVNo.	BrushDustVacuo_D	:=	53	;	//
NameNo.	AnEVNo.	WindDustBlow_D	:=	54	;	//
NameNo.	AnEVNo.	WindDustVacuo_D	:=	55	;	//
NameNo.	AnEVNo.	RJ_Blow	:=	56	;	//
NameNo.	AnEVNo.	RJDustBlow	:=	57	;	//						

